# B&R Automation Studio project DuctLines
Automation Studio 4.2.14.119 SP

## Configuration DUCTO2_RIO

CPU X20CP1584, AutomationRuntime J4.25, Build 4.1.2, Vc V4.25.0, Safety 0.0

### Task classes (Cpu.sw)
```
Cyclic#1 (cycle 1000 us, tolerance 10000 us):
  IMotionCon <- IMotionControl.prg
  CleatRoll <- CleatRoll.prg
Cyclic#2 (cycle 10000 us, tolerance 20000 us):
  PDButtons <- PDButtons.prg
  Uncoiler_2 <- Uncoiler_2.prg
  CoilSelect <- CoilSelect.prg
  MarkTable <- MarkTable.prg
  MarkRF <- MarkRF.prg
  Feeder <- Feeder.prg
  SBrake <- SBrake.prg
  TDCTable <- TDCTable.prg
  TDCRFPshrs <- TDCRFPshrs.prg
  GlueApp <- GlueApp.prg
  Insulmatic <- Insulmatic.prg
  Pinspotter <- Pinspotter.prg
  BrakeCommo <- BrakeCommon.prg
  HydraulicB <- HydraulicBrakeCarriage.prg
  HWBwoPLC <- HWBwoPLC.prg
  MarkHead <- MarkHead.prg
Cyclic#4 (cycle 100000 us, tolerance 100000 us):
  HMIButtons <- HMIButtons.prg
  Server <- LibAsTCP1_ST.Server.prg
Binaries: TCData, arconfig, asfw, ashwd, iomap, User, Role, sysconf
Libraries: standard, MestekLib, AsTCP, runtime, asstring, asieccon, astime
```

### Hardware
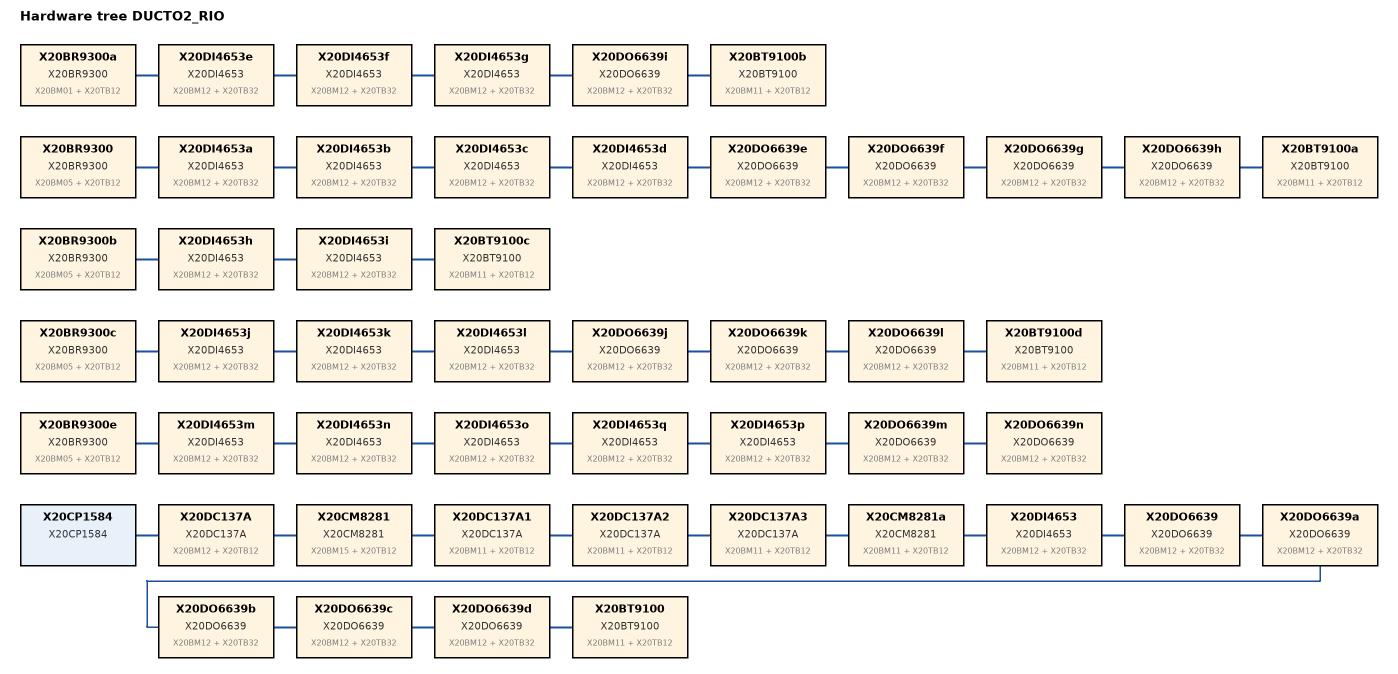
```
X20BM01 : X20BM01 v1.0.1.1
X20BM05 : X20BM05 v1.0.0.3
X20BM05b : X20BM05 v1.0.0.3
X20BM05c : X20BM05 v1.0.0.3
X20BM05d : X20BM05 v1.0.0.3
X20BM11 : X20BM11 v1.0.0.1  [X2X1 -> X20BM12f.X2X2]
X20BM11a : X20BM11 v1.0.0.1  [X2X1 -> X20BM11b.X2X2]
X20BM11b : X20BM11 v1.0.0.1  [X2X1 -> X20BM15.X2X2]
X20BM11c : X20BM11 v1.0.0.1  [X2X1 -> X20BM11a.X2X2]
X20BM11d : X20BM11 v1.0.0.1  [X2X1 -> X20BM11c.X2X2]
X20BM11e : X20BM11 v1.0.0.1  [X2X1 -> X20BM12n.X2X2]
X20BM11f : X20BM11 v1.0.0.1  [X2X1 -> X20BM12r.X2X2]
X20BM11g : X20BM11 v1.0.0.1  [X2X1 -> X20BM12t.X2X2]
X20BM11h : X20BM11 v1.0.0.1  [X2X1 -> X20BM12z.X2X2]
X20BM12 : X20BM12 v1.0.0.1  [X2X1 -> X20BM11d.X2X2]
X20BM12a : X20BM12 v1.0.0.1  [X2X1 -> X20CP1584.IF6]
X20BM12aa : X20BM12 v1.0.0.1  [X2X1 -> X20BM05d.X2X2]
X20BM12ab : X20BM12 v1.0.0.1  [X2X1 -> X20BM12aa.X2X2]
X20BM12ac : X20BM12 v1.0.0.1  [X2X1 -> X20BM12ab.X2X2]
X20BM12ad : X20BM12 v1.0.0.1  [X2X1 -> X20BM12ag.X2X2]
X20BM12ae : X20BM12 v1.0.0.1  [X2X1 -> X20BM12ad.X2X2]
X20BM12af : X20BM12 v1.0.0.1  [X2X1 -> X20BM12ae.X2X2]
X20BM12ag : X20BM12 v1.0.0.1  [X2X1 -> X20BM12ac.X2X2]
X20BM12b : X20BM12 v1.0.0.1  [X2X1 -> X20BM12.X2X2]
X20BM12c : X20BM12 v1.0.0.1  [X2X1 -> X20BM12b.X2X2]
X20BM12d : X20BM12 v1.0.0.1  [X2X1 -> X20BM12c.X2X2]
X20BM12e : X20BM12 v1.0.0.1  [X2X1 -> X20BM12d.X2X2]
X20BM12f : X20BM12 v1.0.0.1  [X2X1 -> X20BM12e.X2X2]
X20BM12g : X20BM12 v1.0.0.1  [X2X1 -> X20BM05.X2X2]
X20BM12h : X20BM12 v1.0.0.1  [X2X1 -> X20BM12g.X2X2]
X20BM12i : X20BM12 v1.0.0.1  [X2X1 -> X20BM12h.X2X2]
X20BM12j : X20BM12 v1.0.0.1  [X2X1 -> X20BM12i.X2X2]
X20BM12k : X20BM12 v1.0.0.1  [X2X1 -> X20BM12j.X2X2]
X20BM12l : X20BM12 v1.0.0.1  [X2X1 -> X20BM12k.X2X2]
X20BM12m : X20BM12 v1.0.0.1  [X2X1 -> X20BM12l.X2X2]
X20BM12n : X20BM12 v1.0.0.1  [X2X1 -> X20BM12m.X2X2]
X20BM12o : X20BM12 v1.0.0.1  [X2X1 -> X20BM01.X2X2]
X20BM12p : X20BM12 v1.0.0.1  [X2X1 -> X20BM12o.X2X2]
X20BM12q : X20BM12 v1.0.0.1  [X2X1 -> X20BM12p.X2X2]
X20BM12r : X20BM12 v1.0.0.1  [X2X1 -> X20BM12q.X2X2]
X20BM12s : X20BM12 v1.0.0.1  [X2X1 -> X20BM05b.X2X2]
X20BM12t : X20BM12 v1.0.0.1  [X2X1 -> X20BM12s.X2X2]
X20BM12u : X20BM12 v1.0.0.1  [X2X1 -> X20BM05c.X2X2]
X20BM12v : X20BM12 v1.0.0.1  [X2X1 -> X20BM12u.X2X2]
X20BM12w : X20BM12 v1.0.0.1  [X2X1 -> X20BM12v.X2X2]
X20BM12x : X20BM12 v1.0.0.1  [X2X1 -> X20BM12w.X2X2]
X20BM12y : X20BM12 v1.0.0.1  [X2X1 -> X20BM12x.X2X2]
X20BM12z : X20BM12 v1.0.0.1  [X2X1 -> X20BM12y.X2X2]
X20BM15 : X20BM15 v1.0.1.0  [X2X1 -> X20BM12a.X2X2 (NodeNumber=2)]
X20BR9300 : X20BR9300 v1.0.3.0  [SS1 -> X20TB12g.SS; SL -> X20BM05.SL1; X2X1 -> X20BT9100.X2X1 (NodeNumber=20)]
  Supervision = off
X20BR9300a : X20BR9300 v1.0.3.0  [SS1 -> X20TB12i.SS; SL -> X20BM01.SL1; X2X1 -> X20BT9100a.X2X1]
  Supervision = off
X20BR9300b : X20BR9300 v1.0.3.0  [SS1 -> X20TB12k.SS; SL -> X20BM05b.SL1; X2X1 -> X20BT9100b.X2X1 (NodeNumber=40)]
  Supervision = off
X20BR9300c : X20BR9300 v1.0.3.0  [SS1 -> X20TB12m.SS; SL -> X20BM05c.SL1; X2X1 -> X20BT9100c.X2X1 (NodeNumber=50)]
  Supervision = off
X20BR9300e : X20BR9300 v1.0.3.0  [SS1 -> X20TB12p.SS; SL -> X20BM05d.SL1; X2X1 -> X20BT9100d.X2X1 (NodeNumber=60)]
  Supervision = off
X20BT9100 : X20BT9100 v1.0.2.4  [SS1 -> X20TB12f.SS; SL -> X20BM11.SL1]
  Supervision = off
X20BT9100a : X20BT9100 v1.0.2.4  [SS1 -> X20TB12h.SS; SL -> X20BM11e.SL1]
  Supervision = off
X20BT9100b : X20BT9100 v1.0.2.4  [SS1 -> X20TB12j.SS; SL -> X20BM11f.SL1]
  Supervision = off
X20BT9100c : X20BT9100 v1.0.2.4  [SS1 -> X20TB12l.SS; SL -> X20BM11g.SL1]
  Supervision = off
X20BT9100d : X20BT9100 v1.0.2.4  [SS1 -> X20TB12n.SS; SL -> X20BM11h.SL1]
  Supervision = off
X20CM8281 : X20CM8281 v1.0.4.0  [SS1 -> X20TB12.SS; SL -> X20BM15.SL1]
  Supervision = off
X20CM8281a : X20CM8281 v1.0.4.0  [SS1 -> X20TB12e.SS; SL -> X20BM11d.SL1]
  Supervision = off
X20CP1584 : X20CP1584 v1.3.0.0
  Connector IF2:
    ActivateDevice = 1
    EthInterfaceRedundant = 0
    Mode = Manual
    InternetAddress = 10.1.254.101
  Connector IF3:
    EplInterfaceRedundant = 0
    EplEthInterfaceRedundant = 0
  ConfigurationID = X20_CPU_test
  EnableUsbRemoteInstall = 1
  TimerDeviceType = SWIOTIMER
  Cyclic1Duration = 1000
  Cyclic1Tolerance = 10000
  Cyclic2Duration = 10000
  Cyclic2Tolerance = 20000
  Cyclic3Duration = 50000
  Cyclic3Tolerance = 50000
  Cyclic4Duration = 100000
  Cyclic4Tolerance = 100000
  Cyclic5Duration = 200000
  Cyclic5Tolerance = 200000
  Cyclic6Duration = 500000
  Cyclic6Tolerance = 500000
  Cyclic7Duration = 1000000
  Cyclic7Tolerance = 1000000
  Cyclic8Duration = 10000
  Cyclic8Tolerance = 30000000
X20DC137A : X20DC137A v1.0.0.3 (LastFrozenVersion=1.0.0.3)  [SS1 -> X20TB12b.SS; SL -> X20BM12a.SL1]
  Supervision = off
  CounterStd01 = 32Bit
  BWConfigChannel03 = off
X20DC137A1 : X20DC137A v1.0.0.3 (LastFrozenVersion=1.0.0.3)  [SS1 -> X20TB12c.SS; SL -> X20BM11b.SL1]
  Supervision = off
  CounterStd01 = 32Bit
  BWConfigChannel03 = off
X20DC137A2 : X20DC137A v1.0.0.3 (LastFrozenVersion=1.0.0.3)  [SS1 -> X20TB12a.SS; SL -> X20BM11a.SL1]
  Supervision = off
  CounterStd01 = 32Bit
  BWConfigChannel03 = off
X20DC137A3 : X20DC137A v1.0.0.3 (LastFrozenVersion=1.0.0.3)  [SS1 -> X20TB12d.SS; SL -> X20BM11c.SL1]
  Supervision = off
  CounterStd01 = 32Bit
  BWConfigChannel03 = off
X20DI4653 : X20DI4653 v1.0.2.0  [SS1 -> X20TB32.SS; SL -> X20BM12.SL1]
  Supervision = off
X20DI4653a : X20DI4653 v1.0.2.0  [SS1 -> X20TB32f.SS; SL -> X20BM12g.SL1]
  Supervision = off
X20DI4653b : X20DI4653 v1.0.2.0  [SS1 -> X20TB32g.SS; SL -> X20BM12h.SL1]
  Supervision = off
X20DI4653c : X20DI4653 v1.0.2.0  [SS1 -> X20TB32h.SS; SL -> X20BM12i.SL1]
  Supervision = off
X20DI4653d : X20DI4653 v1.0.2.0  [SS1 -> X20TB32i.SS; SL -> X20BM12j.SL1]
  Supervision = off
X20DI4653e : X20DI4653 v1.0.2.0  [SS1 -> X20TB32n.SS; SL -> X20BM12o.SL1]
  Supervision = off
X20DI4653f : X20DI4653 v1.0.2.0  [SS1 -> X20TB32o.SS; SL -> X20BM12p.SL1]
  Supervision = off
X20DI4653g : X20DI4653 v1.0.2.0  [SS1 -> X20TB32p.SS; SL -> X20BM12q.SL1]
  Supervision = off
X20DI4653h : X20DI4653 v1.0.2.0  [SS1 -> X20TB32r.SS; SL -> X20BM12s.SL1]
  Supervision = off
X20DI4653i : X20DI4653 v1.0.2.0  [SS1 -> X20TB32s.SS; SL -> X20BM12t.SL1]
  Supervision = off
X20DI4653j : X20DI4653 v1.0.2.0  [SS1 -> X20TB32t.SS; SL -> X20BM12u.SL1]
  Supervision = off
X20DI4653k : X20DI4653 v1.0.2.0  [SS1 -> X20TB32u.SS; SL -> X20BM12v.SL1]
  Supervision = off
X20DI4653l : X20DI4653 v1.0.2.0  [SS1 -> X20TB32v.SS; SL -> X20BM12w.SL1]
  Supervision = off
X20DI4653m : X20DI4653 v1.0.2.0  [SS1 -> X20TB32z.SS; SL -> X20BM12aa.SL1]
  Supervision = off
X20DI4653n : X20DI4653 v1.0.2.0  [SS1 -> X20TB32aa.SS; SL -> X20BM12ab.SL1]
  Supervision = off
X20DI4653o : X20DI4653 v1.0.2.0  [SS1 -> X20TB32ab.SS; SL -> X20BM12ac.SL1]
  Supervision = off
X20DI4653p : X20DI4653 v1.0.2.0  [SS1 -> X20TB32ac.SS; SL -> X20BM12ad.SL1]
  Supervision = off
X20DI4653q : X20DI4653 v1.0.2.0  [SS1 -> X20TB32af.SS; SL -> X20BM12ag.SL1]
  Supervision = off
X20DO6639 : X20DO6639 v1.0.1.0  [SS1 -> X20TB32a.SS; SL -> X20BM12b.SL1]
  Supervision = off
X20DO6639a : X20DO6639 v1.0.1.0  [SS1 -> X20TB32b.SS; SL -> X20BM12c.SL1]
  Supervision = off
X20DO6639b : X20DO6639 v1.0.1.0  [SS1 -> X20TB32c.SS; SL -> X20BM12d.SL1]
  Supervision = off
X20DO6639c : X20DO6639 v1.0.1.0  [SS1 -> X20TB32d.SS; SL -> X20BM12e.SL1]
  Supervision = off
X20DO6639d : X20DO6639 v1.0.1.0  [SS1 -> X20TB32e.SS; SL -> X20BM12f.SL1]
  Supervision = off
X20DO6639e : X20DO6639 v1.0.1.0  [SS1 -> X20TB32j.SS; SL -> X20BM12k.SL1]
  Supervision = off
X20DO6639f : X20DO6639 v1.0.1.0  [SS1 -> X20TB32k.SS; SL -> X20BM12l.SL1]
  Supervision = off
X20DO6639g : X20DO6639 v1.0.1.0  [SS1 -> X20TB32l.SS; SL -> X20BM12m.SL1]
  Supervision = off
X20DO6639h : X20DO6639 v1.0.1.0  [SS1 -> X20TB32m.SS; SL -> X20BM12n.SL1]
  Supervision = off
X20DO6639i : X20DO6639 v1.0.1.0  [SS1 -> X20TB32q.SS; SL -> X20BM12r.SL1]
  Supervision = off
X20DO6639j : X20DO6639 v1.0.1.0  [SS1 -> X20TB32w.SS; SL -> X20BM12x.SL1]
  Supervision = off
X20DO6639k : X20DO6639 v1.0.1.0  [SS1 -> X20TB32x.SS; SL -> X20BM12y.SL1]
  Supervision = off
X20DO6639l : X20DO6639 v1.0.1.0  [SS1 -> X20TB32y.SS; SL -> X20BM12z.SL1]
  Supervision = off
X20DO6639m : X20DO6639 v1.0.1.0  [SS1 -> X20TB32ad.SS; SL -> X20BM12ae.SL1]
  Supervision = off
X20DO6639n : X20DO6639 v1.0.1.0  [SS1 -> X20TB32ae.SS; SL -> X20BM12af.SL1]
  Supervision = off
X20TB12 : X20TB12 v1.0.0.0
X20TB12a : X20TB12 v1.0.0.0
X20TB12b : X20TB12 v1.0.0.0
X20TB12c : X20TB12 v1.0.0.0
X20TB12d : X20TB12 v1.0.0.0
X20TB12e : X20TB12 v1.0.0.0
X20TB12f : X20TB12 v1.0.0.0
X20TB12g : X20TB12 v1.0.0.0
X20TB12h : X20TB12 v1.0.0.0
X20TB12i : X20TB12 v1.0.0.0
X20TB12j : X20TB12 v1.0.0.0
X20TB12k : X20TB12 v1.0.0.0
X20TB12l : X20TB12 v1.0.0.0
X20TB12m : X20TB12 v1.0.0.0
X20TB12n : X20TB12 v1.0.0.0
X20TB12p : X20TB12 v1.0.0.0
X20TB32 : X20TB32 v1.0.0.1
X20TB32a : X20TB32 v1.0.0.1
X20TB32aa : X20TB32 v1.0.0.1
X20TB32ab : X20TB32 v1.0.0.1
X20TB32ac : X20TB32 v1.0.0.1
X20TB32ad : X20TB32 v1.0.0.1
X20TB32ae : X20TB32 v1.0.0.1
X20TB32af : X20TB32 v1.0.0.1
X20TB32b : X20TB32 v1.0.0.1
X20TB32c : X20TB32 v1.0.0.1
X20TB32d : X20TB32 v1.0.0.1
X20TB32e : X20TB32 v1.0.0.1
X20TB32f : X20TB32 v1.0.0.1
X20TB32g : X20TB32 v1.0.0.1
X20TB32h : X20TB32 v1.0.0.1
X20TB32i : X20TB32 v1.0.0.1
X20TB32j : X20TB32 v1.0.0.1
X20TB32k : X20TB32 v1.0.0.1
X20TB32l : X20TB32 v1.0.0.1
X20TB32m : X20TB32 v1.0.0.1
X20TB32n : X20TB32 v1.0.0.1
X20TB32o : X20TB32 v1.0.0.1
X20TB32p : X20TB32 v1.0.0.1
X20TB32q : X20TB32 v1.0.0.1
X20TB32r : X20TB32 v1.0.0.1
X20TB32s : X20TB32 v1.0.0.1
X20TB32t : X20TB32 v1.0.0.1
X20TB32u : X20TB32 v1.0.0.1
X20TB32v : X20TB32 v1.0.0.1
X20TB32w : X20TB32 v1.0.0.1
X20TB32x : X20TB32 v1.0.0.1
X20TB32y : X20TB32 v1.0.0.1
X20TB32z : X20TB32 v1.0.0.1
```

### IoMap.iom - X20CP1584/IoMap.iom
```iecst
VAR_CONFIG
	Cyclic#1.ActlMetalEncoder AT %ID."X20DC137A".Encoder01;
	Cyclic#1.::ProcessorEncoderReset AT %QX."X20DC137A".Encoder01Reset;
	Cyclic#1.ActualDAC1 AT %QW."X20CM8281".AnalogOutput01;
	Cyclic#1.ElectricDriveEnable AT %QX."X20CM8281".DigitalOutput01;
	Cyclic#2.MarkEncoderResetSignal AT %QX."X20DC137A1".Encoder01Reset;
	Cyclic#2.RawMarkEncoder AT %ID."X20DC137A1".Encoder01;
	Cyclic#2.PinspotEncoder AT %ID."X20DC137A2".Encoder01;
	Cyclic#2.PinspotEncoderResetSignal AT %QX."X20DC137A2".Encoder01Reset;
	Cyclic#2.::BrakeEncoderReset AT %QX."X20DC137A3".Encoder01Reset;
	Cyclic#2.BrakeEncoder AT %ID."X20DC137A3".Encoder01;
	Cyclic#2.EStopClear AT %IX."X20DI4653".DigitalInput01;
	Cyclic#2.::PowerOn AT %IX."X20DI4653".DigitalInput02;
	Cyclic#2.doCoilSelect AT %QX."X20DO6639".DigitalOutput01;
	Cyclic#2.doProDuctHydraulics AT %QX."X20DO6639".DigitalOutput02;
	Cyclic#2.BrakeHydraulics AT %QX."X20DO6639".DigitalOutput03;
	Cyclic#2.::MarkTableFwd AT %QX."X20DO6639".DigitalOutput04;
	Cyclic#2.::MarkPshrFwd AT %QX."X20DO6639".DigitalOutput05;
	Cyclic#2.::MarkPusherReverse AT %QX."X20DO6639".DigitalOutput06;
	Cyclic#2.::MarkRollformerOn AT %QX."X20DO6639a".DigitalOutput01;
	Cyclic#2.::TDCConveyorRun AT %QX."X20DO6639a".DigitalOutput02;
	Cyclic#2.::TDCTablePusherFwd AT %QX."X20DO6639a".DigitalOutput03;
	Cyclic#2.::TDCTablePusherReverse AT %QX."X20DO6639a".DigitalOutput04;
	Cyclic#2.doTDCAdjustableHeadIn AT %QX."X20DO6639a".DigitalOutput05;
	Cyclic#2.doTDCAdjustableHeadOut AT %QX."X20DO6639a".DigitalOutput06;
	Cyclic#2.doTDCFixedHeadIn AT %QX."X20DO6639b".DigitalOutput01;
	Cyclic#2.doTDCFixedHeadOut AT %QX."X20DO6639b".DigitalOutput02;
	Cyclic#2.::TDCRFMotor AT %QX."X20DO6639b".DigitalOutput03;
	Cyclic#2.::TDCRFPusherFwd AT %QX."X20DO6639b".DigitalOutput04;
	Cyclic#2.::TDCRFPusherRev AT %QX."X20DO6639b".DigitalOutput05;
	Cyclic#2.::InsulmaticEntranceLowSpeed AT %QX."X20DO6639c".DigitalOutput01;
	Cyclic#2.::InsulmaticExitLowSpeed AT %QX."X20DO6639c".DigitalOutput02;
	Cyclic#2.::InsulmaticExitHiSpeed AT %QX."X20DO6639c".DigitalOutput03;
	Cyclic#2.::InsulmaticEntranceHiSpeed AT %QX."X20DO6639c".DigitalOutput04;
	Cyclic#2.::BrakeConveyorLow AT %QX."X20DO6639c".DigitalOutput05;
	Cyclic#2.::BrakeConveyorHigh AT %QX."X20DO6639c".DigitalOutput06;
	Cyclic#2.::AmberLight AT %QX."X20DO6639d".DigitalOutput01;
	Cyclic#2.::BlueLight AT %QX."X20DO6639d".DigitalOutput02;
	Cyclic#2.::WarningHorn AT %QX."X20DO6639d".DigitalOutput03;
	Cyclic#2.::MarkTableRev AT %QX."X20DO6639d".DigitalOutput04;
	Cyclic#2.::UncoilerJogForwardPB AT %IX."X20DI4653a".DigitalInput01;
	Cyclic#2.::UncoilerJogReversePB AT %IX."X20DI4653a".DigitalInput02;
	Cyclic#2.::SlackBar AT %IX."X20DI4653a".DigitalInput03;
	Cyclic#2.diCoilSelectJog AT %IX."X20DI4653a".DigitalInput04;
	Cyclic#2.::ProcessorJogFwd AT %IX."X20DI4653b".DigitalInput01;
	Cyclic#2.::ProcessorJogRev AT %IX."X20DI4653b".DigitalInput02;
	Cyclic#2.::MatlAtMeasureRoll AT %IX."X20DI4653b".DigitalInput03;
	Cyclic#2.::ShearClampDownProx AT %IX."X20DI4653c".DigitalInput01;
	Cyclic#2.::ShearClampUpProx AT %IX."X20DI4653c".DigitalInput02;
	Cyclic#2.::ShearLeafDownProx AT %IX."X20DI4653c".DigitalInput03;
	Cyclic#2.::ShearLeafUpProx AT %IX."X20DI4653c".DigitalInput04;
	Cyclic#2.::HumpLimitSwitch AT %IX."X20DI4653d".DigitalInput01;
	Cyclic#2.::ShearValve AT %QX."X20DO6639e".DigitalOutput01;
	Cyclic#2.::VValve AT %QX."X20DO6639e".DigitalOutput02;
	Cyclic#2.::LTValve AT %QX."X20DO6639e".DigitalOutput04;
	Cyclic#2.::CenterShuttleOutput AT %QX."X20DO6639e".DigitalOutput05;
	Cyclic#2.::CHoleValve AT %QX."X20DO6639e".DigitalOutput06;
	Cyclic#2.::LeftShuttleOutput AT %QX."X20DO6639f".DigitalOutput01;
	Cyclic#2.::LHoleValve AT %QX."X20DO6639f".DigitalOutput02;
	Cyclic#2.::RightShuttleOutput AT %QX."X20DO6639f".DigitalOutput03;
	Cyclic#2.::RHoleValve AT %QX."X20DO6639f".DigitalOutput04;
	Cyclic#2.::LeftKnockDownRoll AT %QX."X20DO6639f".DigitalOutput05;
	Cyclic#2.::RightKnockDownRoll AT %QX."X20DO6639f".DigitalOutput06;
	Cyclic#2.::ShearClampLowerSolenoid AT %QX."X20DO6639g".DigitalOutput01;
	Cyclic#2.::ShearClampRaiseSolenoid AT %QX."X20DO6639g".DigitalOutput02;
	Cyclic#2.::ShearLeafLowerSolenoid AT %QX."X20DO6639g".DigitalOutput03;
	Cyclic#2.::ShearLeafRaiseSolenoid AT %QX."X20DO6639g".DigitalOutput04;
	Cyclic#2.::SnapLockButtonGag AT %QX."X20DO6639h".DigitalOutput01;
	Cyclic#2.doCoilSelectRollClose AT %QX."X20DO6639h".DigitalOutput02;
	Cyclic#2.::UncoilerRun AT %QX."X20DO6639h".DigitalOutput03;
	Cyclic#2.::UncoilerForwardSolenoid AT %QX."X20DO6639h".DigitalOutput04;
	Cyclic#2.::UncoilerReverseSolenoid AT %QX."X20DO6639h".DigitalOutput05;
	Cyclic#2.diFeedInitButton AT %IX."X20DI4653f".DigitalInput01;
	Cyclic#2.::TDCTablePartProx AT %IX."X20DI4653f".DigitalInput02;
	Cyclic#2.::TDCTablePause AT %IX."X20DI4653f".DigitalInput03;
	Cyclic#2.::TDCTablePushStop AT %IX."X20DI4653f".DigitalInput04;
	Cyclic#2.::TDCTablePusherRevPB AT %IX."X20DI4653g".DigitalInput01;
	Cyclic#2.::diMarkHeadUpProx AT %IX."X20DI4653g".DigitalInput02;
	Cyclic#2.::diMarkHeadDownProx AT %IX."X20DI4653g".DigitalInput03;
	Cyclic#2.::MarkGateRaise AT %QX."X20DO6639i".DigitalOutput01;
	Cyclic#2.doMarkRollformerHeadLower AT %QX."X20DO6639i".DigitalOutput02;
	Cyclic#2.doMarkRollformerHeadRaise AT %QX."X20DO6639i".DigitalOutput03;
	Cyclic#2.diTDCFixedHeadJogIn AT %IX."X20DI4653h".DigitalInput01;
	Cyclic#2.diTDCFixedHeadJogOut AT %IX."X20DI4653h".DigitalInput02;
	Cyclic#2.diTDCAdjustableHeadJogIn AT %IX."X20DI4653h".DigitalInput03;
	Cyclic#2.diTDCAdjustableHeadJogOut AT %IX."X20DI4653h".DigitalInput04;
	Cyclic#2.::diTDCRollformerJog AT %IX."X20DI4653i".DigitalInput01;
	Cyclic#2.::TDCPushStrokeComplete AT %IX."X20DI4653i".DigitalInput03;
	Cyclic#2.::TDCPusherRevPB AT %IX."X20DI4653i".DigitalInput04;
	Cyclic#2.::GluePartSense AT %IX."X20DI4653j".DigitalInput01;
	Cyclic#2.::RaiseImaticBlade AT %IX."X20DI4653k".DigitalInput01;
	Cyclic#2.::InsulationFeed AT %IX."X20DI4653k".DigitalInput02;
	Cyclic#2.::ISquarePinOn AT %IX."X20DI4653k".DigitalInput03;
	Cyclic#2.::PartAtISquarePin AT %IX."X20DI4653k".DigitalInput04;
	Cyclic#2.::PartAtInsulationFeed AT %IX."X20DI4653l".DigitalInput01;
	Cyclic#2.::PartPresentPSpotter AT %IX."X20DI4653l".DigitalInput02;
	Cyclic#2.::GlueSprayEnable AT %QX."X20DO6639j".DigitalOutput03;
	Cyclic#2.::ImaticFeedRoll AT %QX."X20DO6639k".DigitalOutput03;
	Cyclic#2.::ImaticPressRoll AT %QX."X20DO6639k".DigitalOutput04;
	Cyclic#2.::ImaticSquarePin AT %QX."X20DO6639k".DigitalOutput05;
	Cyclic#2.::ImaticBladeUp AT %QX."X20DO6639l".DigitalOutput01;
	Cyclic#2.::ImaticBladeDown AT %QX."X20DO6639l".DigitalOutput02;
	Cyclic#2.::PinspotterDrive AT %QX."X20DO6639l".DigitalOutput03;
	Cyclic#2.::CarriageReference AT %IX."X20DI4653m".DigitalInput01;
	Cyclic#2.::BrakeArmLwrInhibit AT %IX."X20DI4653m".DigitalInput02;
	Cyclic#2.::BrakeBeamLwrInhibit AT %IX."X20DI4653m".DigitalInput03;
	Cyclic#2.::EjectComplete AT %IX."X20DI4653m".DigitalInput04;
	Cyclic#2.::BrakeLeafHomeProx AT %IX."X20DI4653n".DigitalInput01;
	Cyclic#2.::BrakeBeamDownProx AT %IX."X20DI4653n".DigitalInput02;
	Cyclic#2.::BrakeBeamUpProx AT %IX."X20DI4653n".DigitalInput03;
	Cyclic#2.diWBrakeArmsUp AT %IX."X20DI4653n".DigitalInput04;
	Cyclic#2.::BrakePartPresent AT %IX."X20DI4653o".DigitalInput01;
	Cyclic#2.::MaterialClamped AT %IX."X20DI4653o".DigitalInput02;
	Cyclic#2.BrakeManualButton AT %IX."X20DI4653o".DigitalInput04;
	Cyclic#2.::BrakeSingleCycle AT %IX."X20DI4653p".DigitalInput01;
	Cyclic#2.::MoveToBeam AT %QX."X20DO6639m".DigitalOutput01;
	Cyclic#2.::MoveAwayBeam AT %QX."X20DO6639m".DigitalOutput02;
	Cyclic#2.::BrakeHighSpeedRelay AT %QX."X20DO6639m".DigitalOutput03;
	Cyclic#2.::CarriageArmRaise AT %QX."X20DO6639m".DigitalOutput04;
	Cyclic#2.::CarriageArmLower AT %QX."X20DO6639m".DigitalOutput05;
	Cyclic#2.::CarriageClampClose AT %QX."X20DO6639m".DigitalOutput06;
	Cyclic#2.::BrakeBeamRaise AT %QX."X20DO6639n".DigitalOutput01;
	Cyclic#2.::BrakeBeamLower AT %QX."X20DO6639n".DigitalOutput02;
	Cyclic#2.::BrakeLeafRaise AT %QX."X20DO6639n".DigitalOutput03;
	Cyclic#2.::BrakeLeafLower AT %QX."X20DO6639n".DigitalOutput04;
	Cyclic#2.::BrakeManualIndicator AT %QX."X20DO6639n".DigitalOutput05;
	Cyclic#2.::BrakeAutoIndicator AT %QX."X20DO6639n".DigitalOutput06;
	Cyclic#2.::BrakeAutoButton AT %IX."X20DI4653q".DigitalInput01;
	Cyclic#2.diBrakeCarriageJogIn AT %IX."X20DI4653q".DigitalInput02;
	Cyclic#2.diBrakeCarriageJogOut AT %IX."X20DI4653q".DigitalInput03;
	Cyclic#2.::BrakeSequenceReset AT %IX."X20DI4653q".DigitalInput04;
	Cyclic#2.::MatlAtMarkTable AT %IX."X20DI4653e".DigitalInput01;
	Cyclic#2.::MarkPushComplete AT %IX."X20DI4653e".DigitalInput02;
	Cyclic#2.::MarkPusherStop AT %IX."X20DI4653e".DigitalInput03;
	Cyclic#2.::MarkTTPusherJogRevPB AT %IX."X20DI4653e".DigitalInput04;
END_VAR
```

## Configuration DUCTO2_V02

CPU X20CP1584, AutomationRuntime J4.25, Build 4.1.2, Vc V4.25.0, Safety 0.0

### Hardware
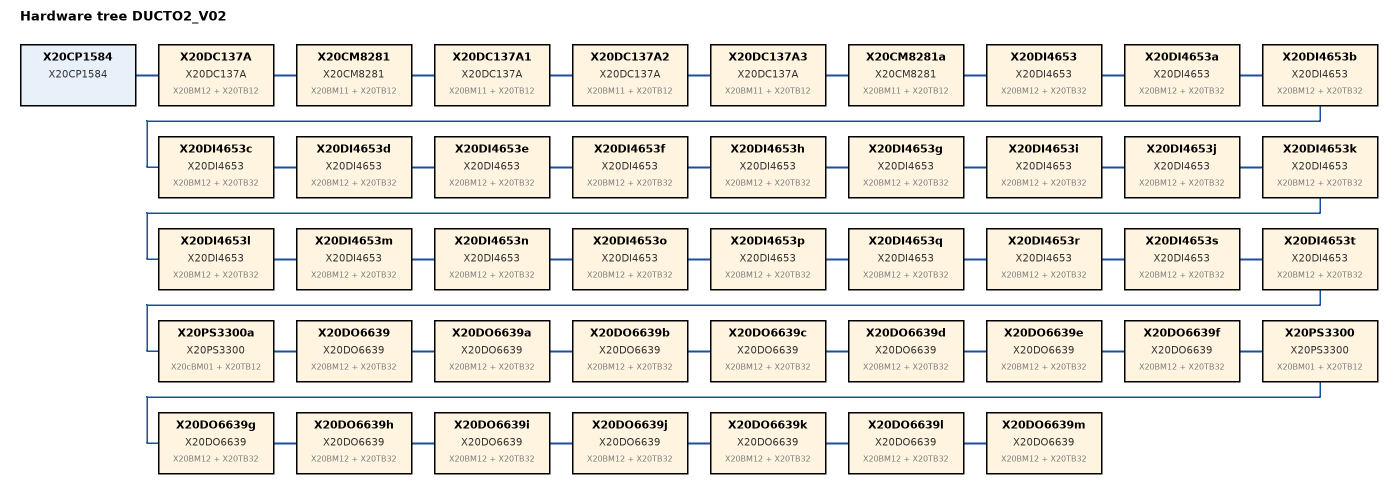
```
X20BM01 : X20BM01 v1.0.1.1  [X2X1 -> X20BM12ab.X2X2]
X20BM11 : X20BM11 v1.0.0.1  [X2X1 -> X20BM12a.X2X2]
X20BM11a : X20BM11 v1.0.0.1  [X2X1 -> X20BM11b.X2X2]
X20BM11b : X20BM11 v1.0.0.1  [X2X1 -> X20BM11.X2X2]
X20BM11c : X20BM11 v1.0.0.1  [X2X1 -> X20BM11a.X2X2]
X20BM11d : X20BM11 v1.0.0.1  [X2X1 -> X20BM11c.X2X2]
X20BM12 : X20BM12 v1.0.0.1  [X2X1 -> X20BM11d.X2X2]
X20BM12a : X20BM12 v1.0.0.1  [X2X1 -> X20CP1584.IF6]
X20BM12aa : X20BM12 v1.0.0.1  [X2X1 -> X20BM12z.X2X2]
X20BM12ab : X20BM12 v1.0.0.1  [X2X1 -> X20BM12aa.X2X2]
X20BM12ac : X20BM12 v1.0.0.1  [X2X1 -> X20BM01.X2X2]
X20BM12ad : X20BM12 v1.0.0.1  [X2X1 -> X20BM12ac.X2X2]
X20BM12ae : X20BM12 v1.0.0.1  [X2X1 -> X20BM12ad.X2X2]
X20BM12af : X20BM12 v1.0.0.1  [X2X1 -> X20BM12ae.X2X2]
X20BM12ag : X20BM12 v1.0.0.1  [X2X1 -> X20BM12af.X2X2]
X20BM12ah : X20BM12 v1.0.0.1  [X2X1 -> X20BM12ag.X2X2]
X20BM12ai : X20BM12 v1.0.0.1  [X2X1 -> X20BM12ah.X2X2]
X20BM12b : X20BM12 v1.0.0.1  [X2X1 -> X20BM12.X2X2]
X20BM12c : X20BM12 v1.0.0.1  [X2X1 -> X20BM12b.X2X2]
X20BM12d : X20BM12 v1.0.0.1  [X2X1 -> X20BM12c.X2X2]
X20BM12e : X20BM12 v1.0.0.1  [X2X1 -> X20BM12d.X2X2]
X20BM12f : X20BM12 v1.0.0.1  [X2X1 -> X20BM12e.X2X2]
X20BM12g : X20BM12 v1.0.0.1  [X2X1 -> X20BM12f.X2X2]
X20BM12h : X20BM12 v1.0.0.1  [X2X1 -> X20BM12i.X2X2]
X20BM12i : X20BM12 v1.0.0.1  [X2X1 -> X20BM12g.X2X2]
X20BM12j : X20BM12 v1.0.0.1  [X2X1 -> X20BM12h.X2X2]
X20BM12k : X20BM12 v1.0.0.1  [X2X1 -> X20BM12j.X2X2]
X20BM12l : X20BM12 v1.0.0.1  [X2X1 -> X20BM12k.X2X2]
X20BM12m : X20BM12 v1.0.0.1  [X2X1 -> X20BM12l.X2X2]
X20BM12n : X20BM12 v1.0.0.1  [X2X1 -> X20BM12m.X2X2]
X20BM12o : X20BM12 v1.0.0.1  [X2X1 -> X20BM12n.X2X2]
X20BM12p : X20BM12 v1.0.0.1  [X2X1 -> X20BM12o.X2X2]
X20BM12q : X20BM12 v1.0.0.1  [X2X1 -> X20BM12p.X2X2]
X20BM12r : X20BM12 v1.0.0.1  [X2X1 -> X20BM12q.X2X2]
X20BM12s : X20BM12 v1.0.0.1  [X2X1 -> X20BM12r.X2X2]
X20BM12t : X20BM12 v1.0.0.1  [X2X1 -> X20BM12s.X2X2]
X20BM12u : X20BM12 v1.0.0.1  [X2X1 -> X20BM12t.X2X2]
X20BM12v : X20BM12 v1.0.0.1  [X2X1 -> X20cBM01.X2X2]
X20BM12w : X20BM12 v1.0.0.1  [X2X1 -> X20BM12v.X2X2]
X20BM12x : X20BM12 v1.0.0.1  [X2X1 -> X20BM12w.X2X2]
X20BM12y : X20BM12 v1.0.0.1  [X2X1 -> X20BM12x.X2X2]
X20BM12z : X20BM12 v1.0.0.1  [X2X1 -> X20BM12y.X2X2]
X20CM8281 : X20CM8281 v1.0.4.0  [SS1 -> X20TB12.SS; SL -> X20BM11.SL1]
  Supervision = off
X20CM8281a : X20CM8281 v1.0.4.0  [SS1 -> X20TB12e.SS; SL -> X20BM11d.SL1]
  Supervision = off
X20CP1584 : X20CP1584 v1.3.0.0
  Connector IF2:
    ActivateDevice = 1
    EthInterfaceRedundant = 0
    Mode = Manual
    InternetAddress = 10.1.254.101
  Connector IF3:
    EplInterfaceRedundant = 0
    CycleTime = 1000
    EplEthInterfaceRedundant = 0
  Connector IF6:
    CycleTime = 1000
  ConfigurationID = X20_CPU_test
  PermanentPvSize = 4096
  EnableUsbRemoteInstall = 1
  TimerDeviceType = EPLX2X
  Cyclic1Duration = 1000
  Cyclic1Tolerance = 0
  Cyclic1Output = 1
  Cyclic2Duration = 20000
  Cyclic2Tolerance = 20000
  Cyclic3Duration = 50000
  Cyclic3Tolerance = 50000
  Cyclic4Duration = 100000
  Cyclic4Tolerance = 100000
  Cyclic5Duration = 200000
  Cyclic5Tolerance = 200000
  Cyclic6Duration = 500000
  Cyclic6Tolerance = 500000
  Cyclic7Duration = 1000000
  Cyclic7Tolerance = 1000000
  Cyclic8Duration = 10000
  Cyclic8Tolerance = 30000000
  TimerDevice = X20CP1584.IF6
X20DC137A : X20DC137A v1.0.0.3  [SS1 -> X20TB12b.SS; SL -> X20BM12a.SL1]
  Supervision = off
  CounterStd01 = 32Bit
  BWConfigChannel03 = off
X20DC137A1 : X20DC137A v1.0.0.3  [SS1 -> X20TB12c.SS; SL -> X20BM11b.SL1]
  Supervision = off
  CounterStd01 = 32Bit
  BWConfigChannel03 = off
X20DC137A2 : X20DC137A v1.0.0.3  [SS1 -> X20TB12a.SS; SL -> X20BM11a.SL1]
  Supervision = off
  CounterStd01 = 32Bit
  BWConfigChannel03 = off
X20DC137A3 : X20DC137A v1.0.0.3  [SS1 -> X20TB12d.SS; SL -> X20BM11c.SL1]
  Supervision = off
  CounterStd01 = 32Bit
  BWConfigChannel03 = off
X20DI4653 : X20DI4653 v1.0.2.0  [SS1 -> X20TB32.SS; SL -> X20BM12.SL1]
  Supervision = off
X20DI4653a : X20DI4653 v1.0.2.0  [SS1 -> X20TB32a.SS; SL -> X20BM12b.SL1]
  Supervision = off
X20DI4653b : X20DI4653 v1.0.2.0  [SS1 -> X20TB32b.SS; SL -> X20BM12c.SL1]
  Supervision = off
X20DI4653c : X20DI4653 v1.0.2.0  [SS1 -> X20TB32c.SS; SL -> X20BM12d.SL1]
  Supervision = off
X20DI4653d : X20DI4653 v1.0.2.0  [SS1 -> X20TB32d.SS; SL -> X20BM12e.SL1]
  Supervision = off
X20DI4653e : X20DI4653 v1.0.2.0  [SS1 -> X20TB32e.SS; SL -> X20BM12f.SL1]
  Supervision = off
X20DI4653f : X20DI4653 v1.0.2.0  [SS1 -> X20TB32f.SS; SL -> X20BM12g.SL1]
  Supervision = off
X20DI4653g : X20DI4653 v1.0.2.0  [SS1 -> X20TB32g.SS; SL -> X20BM12h.SL1]
  Supervision = off
X20DI4653h : X20DI4653 v1.0.2.0  [SS1 -> X20TB32h.SS; SL -> X20BM12i.SL1]
  Supervision = off
X20DI4653i : X20DI4653 v1.0.2.0  [SS1 -> X20TB32i.SS; SL -> X20BM12j.SL1]
  Supervision = off
X20DI4653j : X20DI4653 v1.0.2.0  [SS1 -> X20TB32j.SS; SL -> X20BM12k.SL1]
  Supervision = off
X20DI4653k : X20DI4653 v1.0.2.0  [SS1 -> X20TB32k.SS; SL -> X20BM12l.SL1]
  Supervision = off
X20DI4653l : X20DI4653 v1.0.2.0  [SS1 -> X20TB32l.SS; SL -> X20BM12m.SL1]
  Supervision = off
X20DI4653m : X20DI4653 v1.0.2.0  [SS1 -> X20TB32m.SS; SL -> X20BM12n.SL1]
  Supervision = off
X20DI4653n : X20DI4653 v1.0.2.0  [SS1 -> X20TB32n.SS; SL -> X20BM12o.SL1]
  Supervision = off
X20DI4653o : X20DI4653 v1.0.2.0  [SS1 -> X20TB32o.SS; SL -> X20BM12p.SL1]
  Supervision = off
X20DI4653p : X20DI4653 v1.0.2.0  [SS1 -> X20TB32p.SS; SL -> X20BM12q.SL1]
  Supervision = off
X20DI4653q : X20DI4653 v1.0.2.0  [SS1 -> X20TB32q.SS; SL -> X20BM12r.SL1]
  Supervision = off
X20DI4653r : X20DI4653 v1.0.2.0  [SS1 -> X20TB32r.SS; SL -> X20BM12s.SL1]
  Supervision = off
X20DI4653s : X20DI4653 v1.0.2.0  [SS1 -> X20TB32s.SS; SL -> X20BM12t.SL1]
  Supervision = off
X20DI4653t : X20DI4653 v1.0.2.0  [SS1 -> X20TB32t.SS; SL -> X20BM12u.SL1]
  Supervision = off
X20DO6639 : X20DO6639 v1.0.1.0  [SS1 -> X20TB32u.SS; SL -> X20BM12v.SL1]
  Supervision = off
X20DO6639a : X20DO6639 v1.0.1.0  [SS1 -> X20TB32v.SS; SL -> X20BM12w.SL1]
  Supervision = off
X20DO6639b : X20DO6639 v1.0.1.0  [SS1 -> X20TB32w.SS; SL -> X20BM12x.SL1]
  Supervision = off
X20DO6639c : X20DO6639 v1.0.1.0  [SS1 -> X20TB32x.SS; SL -> X20BM12y.SL1]
  Supervision = off
X20DO6639d : X20DO6639 v1.0.1.0  [SS1 -> X20TB32y.SS; SL -> X20BM12z.SL1]
  Supervision = off
X20DO6639e : X20DO6639 v1.0.1.0  [SS1 -> X20TB32z.SS; SL -> X20BM12aa.SL1]
  Supervision = off
X20DO6639f : X20DO6639 v1.0.1.0  [SS1 -> X20TB32aa.SS; SL -> X20BM12ab.SL1]
  Supervision = off
X20DO6639g : X20DO6639 v1.0.1.0  [SS1 -> X20TB32ab.SS; SL -> X20BM12ac.SL1]
  Supervision = off
X20DO6639h : X20DO6639 v1.0.1.0  [SS1 -> X20TB32ac.SS; SL -> X20BM12ad.SL1]
  Supervision = off
X20DO6639i : X20DO6639 v1.0.1.0  [SS1 -> X20TB32ad.SS; SL -> X20BM12ae.SL1]
  Supervision = off
X20DO6639j : X20DO6639 v1.0.1.0  [SS1 -> X20TB32ae.SS; SL -> X20BM12af.SL1]
  Supervision = off
X20DO6639k : X20DO6639 v1.0.1.0  [SS1 -> X20TB32af.SS; SL -> X20BM12ag.SL1]
  Supervision = off
X20DO6639l : X20DO6639 v1.0.1.0  [SS1 -> X20TB32ag.SS; SL -> X20BM12ah.SL1]
  Supervision = off
X20DO6639m : X20DO6639 v1.0.1.0  [SS1 -> X20TB32ah.SS; SL -> X20BM12ai.SL1]
  Supervision = off
X20PS3300 : X20PS3300 v1.1.0.0  [SS1 -> X20TB12g.SS; SL -> X20BM01.SL1]
  Supervision = off
X20PS3300a : X20PS3300 v1.1.0.0  [SS1 -> X20TB12f.SS; SL -> X20cBM01.SL1]
  Supervision = off
X20TB12 : X20TB12 v1.0.0.0
X20TB12a : X20TB12 v1.0.0.0
X20TB12b : X20TB12 v1.0.0.0
X20TB12c : X20TB12 v1.0.0.0
X20TB12d : X20TB12 v1.0.0.0
X20TB12e : X20TB12 v1.0.0.0
X20TB12f : X20TB12 v1.0.0.0
X20TB12g : X20TB12 v1.0.0.0
X20TB32 : X20TB32 v1.0.0.1
X20TB32a : X20TB32 v1.0.0.1
X20TB32aa : X20TB32 v1.0.0.1
X20TB32ab : X20TB32 v1.0.0.1
X20TB32ac : X20TB32 v1.0.0.1
X20TB32ad : X20TB32 v1.0.0.1
X20TB32ae : X20TB32 v1.0.0.1
X20TB32af : X20TB32 v1.0.0.1
X20TB32ag : X20TB32 v1.0.0.1
X20TB32ah : X20TB32 v1.0.0.1
X20TB32b : X20TB32 v1.0.0.1
X20TB32c : X20TB32 v1.0.0.1
X20TB32d : X20TB32 v1.0.0.1
X20TB32e : X20TB32 v1.0.0.1
X20TB32f : X20TB32 v1.0.0.1
X20TB32g : X20TB32 v1.0.0.1
X20TB32h : X20TB32 v1.0.0.1
X20TB32i : X20TB32 v1.0.0.1
X20TB32j : X20TB32 v1.0.0.1
X20TB32k : X20TB32 v1.0.0.1
X20TB32l : X20TB32 v1.0.0.1
X20TB32m : X20TB32 v1.0.0.1
X20TB32n : X20TB32 v1.0.0.1
X20TB32o : X20TB32 v1.0.0.1
X20TB32p : X20TB32 v1.0.0.1
X20TB32q : X20TB32 v1.0.0.1
X20TB32r : X20TB32 v1.0.0.1
X20TB32s : X20TB32 v1.0.0.1
X20TB32t : X20TB32 v1.0.0.1
X20TB32u : X20TB32 v1.0.0.1
X20TB32v : X20TB32 v1.0.0.1
X20TB32w : X20TB32 v1.0.0.1
X20TB32x : X20TB32 v1.0.0.1
X20TB32y : X20TB32 v1.0.0.1
X20TB32z : X20TB32 v1.0.0.1
X20cBM01 : X20cBM01 v1.0.1.0  [X2X1 -> X20BM12u.X2X2]
```

### Cpu.per - X20CP1584/Cpu.per
```iecst
VAR_CONFIG
	MarkEncoder AT %MD0; (* *)
END_VAR
```

### IoMap.iom - X20CP1584/IoMap.iom
```iecst
VAR_CONFIG
	Cyclic#1.ActlMetalEncoder AT %ID."X20DC137A".Encoder01;
	Cyclic#1.ActualDAC1 AT %QW."X20CM8281".AnalogOutput01;
	Cyclic#2.AmberLight AT %QX."X20DO6639".DigitalOutput02;
	Cyclic#2.BatchActivePhysical AT %QX."X20DO6639".DigitalOutput06;
	Cyclic#2.::BrakeEncoderReset AT %QX."X20DC137A3".Encoder01Reset;
	Cyclic#2.BlockingValve AT %QX."X20DO6639".DigitalOutput05;
	Cyclic#2.BlueLight AT %QX."X20DO6639".DigitalOutput03;
	Cyclic#2.BrakeArmLwrInhibit AT %IX."X20DI4653p".DigitalInput02;
	Cyclic#2.BrakeAutoIndicator AT %QX."X20DO6639l".DigitalOutput05;
	Cyclic#2.BrakeAutoRequest AT %IX."X20DI4653s".DigitalInput02;
	Cyclic#2.BrakeBeamDownProx AT %IX."X20DI4653q".DigitalInput02;
	Cyclic#2.BrakeBeamLower AT %QX."X20DO6639l".DigitalOutput02;
	Cyclic#2.BrakeBeamLwrInhibit AT %IX."X20DI4653p".DigitalInput03;
	Cyclic#2.BrakeBeamRaise AT %QX."X20DO6639l".DigitalOutput01;
	Cyclic#2.BrakeBeamUpProx AT %IX."X20DI4653q".DigitalInput03;
	Cyclic#2.BrakeCarriageJogIn AT %IX."X20DI4653s".DigitalInput03;
	Cyclic#2.BrakeCarriageJogOut AT %IX."X20DI4653s".DigitalInput04;
	Cyclic#2.BrakeEncoder AT %ID."X20DC137A3".Encoder01;
	Cyclic#2.BrakeHighSpeedRelay AT %QX."X20DO6639k".DigitalOutput03;
	Cyclic#2.BrakeHydraulics AT %IX."X20DI4653r".DigitalInput03;
	Cyclic#2.BrakeLeafHomeProx AT %IX."X20DI4653q".DigitalInput01;
	Cyclic#2.BrakeLeafLower AT %QX."X20DO6639l".DigitalOutput04;
	Cyclic#2.BrakeLeafRaise AT %QX."X20DO6639l".DigitalOutput03;
	Cyclic#2.BrakeManual AT %IX."X20DI4653s".DigitalInput01;
	Cyclic#2.BrakeOn AT %QX."X20DO6639m".DigitalOutput01;
	Cyclic#2.BrakePartPresent AT %IX."X20DI4653r".DigitalInput01;
	Cyclic#2.BrakeSequenceReset AT %IX."X20DI4653t".DigitalInput01;
	Cyclic#2.BrakeSetButton AT %IX."X20DI4653t".DigitalInput02;
	Cyclic#2.BrakeSingleCycle AT %IX."X20DI4653t".DigitalInput03;
	BrakeSpeedSwitch AT %IX."X20DI4653r".DigitalInput04;
	Cyclic#2.CarriageArmLower AT %QX."X20DO6639k".DigitalOutput05;
	Cyclic#2.CarriageArmRaise AT %QX."X20DO6639k".DigitalOutput04;
	Cyclic#2.CarriageClampClose AT %QX."X20DO6639k".DigitalOutput06;
	Cyclic#2.CarriageReference AT %IX."X20DI4653p".DigitalInput01;
	Cyclic#2.CenterShuttleOutput AT %QX."X20DO6639b".DigitalOutput01;
	Cyclic#2.CHoleValve AT %QX."X20DO6639b".DigitalOutput02;
	Cyclic#2.CleatRollerSheetSense AT %IX."X20DI4653j".DigitalInput03;
	Cyclic#2.DuctoAuto AT %IX."X20DI4653a".DigitalInput01;
	Cyclic#2.DuctSelected AT %IX."X20DI4653e".DigitalInput01;
	Cyclic#2.EjectComplete AT %IX."X20DI4653p".DigitalInput04;
	Cyclic#1.ElectricDriveEnable AT %QX."X20CM8281".DigitalOutput01;
	Cyclic#2.EStopClear AT %IX."X20DI4653".DigitalInput01;
	Cyclic#2.ExitBeltsOn AT %IX."X20DI4653j".DigitalInput01;
	Cyclic#2.FeedInitButton AT %IX."X20DI4653".DigitalInput04;
	Cyclic#2.InsulmaticEntranceHiSpeed AT %QX."X20DO6639m".DigitalOutput04;
	Cyclic#2.InsulmaticEntranceLowSpeed AT %QX."X20DO6639i".DigitalOutput02;
	Cyclic#2.GlueFlushPB AT %IX."X20DI4653l".DigitalInput03;
	Cyclic#2.GluePartSense AT %IX."X20DI4653l".DigitalInput02;
	Cyclic#2.GluePumpOnSwitch AT %IX."X20DI4653l".DigitalInput01;
	Cyclic#2.GlueServiceSwitch AT %IX."X20DI4653m".DigitalInput01;
	Cyclic#2.HumpLimitSwitch AT %IX."X20DI4653c".DigitalInput01;
	Cyclic#2.ImaticBladeDown AT %QX."X20DO6639j".DigitalOutput01;
	Cyclic#2.ImaticBladeUp AT %QX."X20DO6639i".DigitalOutput06;
	Cyclic#2.ImaticFeedRoll AT %QX."X20DO6639i".DigitalOutput03;
	Cyclic#2.ImaticPressRoll AT %QX."X20DO6639i".DigitalOutput04;
	Cyclic#2.::ISquarePinOn AT %IX."X20DI4653n".DigitalInput04;
	Cyclic#2.ImaticSquarePin AT %QX."X20DO6639i".DigitalOutput05;
	Cyclic#2.InsulationFeed AT %IX."X20DI4653n".DigitalInput03;
	Cyclic#2.InsulmaticExitHiSpeed AT %QX."X20DO6639m".DigitalOutput02;
	Cyclic#2.InsulmaticExitLowSpeed AT %QX."X20DO6639m".DigitalOutput03;
	Cyclic#2.InsulmaticOn AT %IX."X20DI4653n".DigitalInput01;
	LBrakePartEjectSolenoid AT %QX."X20DO6639l".DigitalOutput06;
	Cyclic#2.LeftShuttleOutput AT %QX."X20DO6639b".DigitalOutput03;
	Cyclic#2.LHoleValve AT %QX."X20DO6639b".DigitalOutput04;
	Cyclic#2.LTValve AT %QX."X20DO6639a".DigitalOutput04;
	Cyclic#2.MarkAuto AT %IX."X20DI4653d".DigitalInput02;
	Cyclic#2.MarkConveyorDelayFwd AT %IX."X20DI4653i".DigitalInput04;
	Cyclic#2.MarkEncoderResetSignal AT %QX."X20DC137A1".Encoder01Reset;
	Cyclic#2.MarkGateRaise AT %QX."X20DO6639f".DigitalOutput01;
	Cyclic#2.MarkHeadJogInSwitch AT %IX."X20DI4653e".DigitalInput03;
	Cyclic#2.MarkHeadJogOutSwitch AT %IX."X20DI4653e".DigitalInput04;
	Cyclic#2.MarkHiSpeedSignal AT %IX."X20DI4653e".DigitalInput02;
	Cyclic#2.MarkPshrFwd AT %QX."X20DO6639e".DigitalOutput06;
	Cyclic#2.MarkPushComplete AT %IX."X20DI4653h".DigitalInput02;
	Cyclic#2.MarkPusherStop AT %IX."X20DI4653i".DigitalInput01;
	Cyclic#2.MarkRefSwitch AT %IX."X20DI4653f".DigitalInput01;
	Cyclic#2.MarkRFHighSpeed AT %QX."X20DO6639c".DigitalOutput05;
	Cyclic#2.MarkRFMoveIn AT %QX."X20DO6639c".DigitalOutput03;
	Cyclic#2.MarkRFMoveOut AT %QX."X20DO6639c".DigitalOutput04;
	Cyclic#2.MarkRollformerOn AT %IX."X20DI4653d".DigitalInput01;
	Cyclic#2.MarkSetButton AT %IX."X20DI4653d".DigitalInput03;
	Cyclic#2.MarkTableFwd AT %QX."X20DO6639e".DigitalOutput03;
	Cyclic#2.::MarkTableStart AT %IX."X20DI4653g".DigitalInput01;
	Cyclic#2.MarkTableRev AT %QX."X20DO6639e".DigitalOutput04;
	Cyclic#2.MaterialClamped AT %IX."X20DI4653r".DigitalInput02;
	Cyclic#2.MatlAtMarkTable AT %IX."X20DI4653g".DigitalInput03;
	Cyclic#2.MatlAtMeasureRoll AT %IX."X20DI4653a".DigitalInput04;
	Cyclic#2.MoveAwayBeam AT %QX."X20DO6639k".DigitalOutput02;
	Cyclic#2.MoveToBeam AT %QX."X20DO6639k".DigitalOutput01;
	Cyclic#2.MTBlockedValve AT %QX."X20DO6639g".DigitalOutput06;
	Cyclic#2.MTFlushTubeCloseSolenoid AT %QX."X20DO6639h".DigitalOutput01;
	Cyclic#2.MTFlushTubeOpenSolenoid AT %QX."X20DO6639h".DigitalOutput02;
	Cyclic#2.MTGlueValveSolenoid AT %QX."X20DO6639h".DigitalOutput03;
	Cyclic#2.MTPlungerValveSolenoid AT %QX."X20DO6639h".DigitalOutput05;
	Cyclic#2.MTWaterFlushSolenoid AT %QX."X20DO6639h".DigitalOutput04;
	Cyclic#2.MTWaterSupplySolenoid AT %QX."X20DO6639h".DigitalOutput06;
	Cyclic#2.::LeftKnockDownRoll AT %QX."X20DO6639f".DigitalOutput03;
	Cyclic#2.PartAtInsulationFeed AT %IX."X20DI4653o".DigitalInput02;
	Cyclic#2.PartAtISquarePin AT %IX."X20DI4653o".DigitalInput01;
	Cyclic#2.PartPresentPSpotter AT %IX."X20DI4653o".DigitalInput03;
	Cyclic#2.PinspotEncoder AT %ID."X20DC137A2".Encoder01;
	Cyclic#2.PinspotEncoderResetSignal AT %QX."X20DC137A2".Encoder01Reset;
	Cyclic#2.PinspotterDrive AT %QX."X20DO6639j".DigitalOutput02;
	Cyclic#2.PinspotterLoad AT %QX."X20DO6639j".DigitalOutput03;
	Cyclic#2.PowerOn AT %IX."X20DI4653c".DigitalInput04;
	Cyclic#2.ProcessorDriveEnable AT %IX."X20DI4653".DigitalInput03;
	Cyclic#2.ProcessorJogFwd AT %IX."X20DI4653a".DigitalInput02;
	Cyclic#2.ProcessorJogRev AT %IX."X20DI4653a".DigitalInput03;
	Cyclic#2.RaiseImaticBlade AT %IX."X20DI4653n".DigitalInput02;
	Cyclic#2.RawMarkEncoder AT %ID."X20DC137A1".Encoder01;
	Cyclic#2.RHoleValve AT %QX."X20DO6639a".DigitalOutput06;
	Cyclic#2.RightShuttleOutput AT %QX."X20DO6639a".DigitalOutput05;
	Cyclic#2.ShearClampDownProx AT %IX."X20DI4653b".DigitalInput01;
	Cyclic#2.ShearClampLowerSolenoid AT %QX."X20DO6639b".DigitalOutput05;
	Cyclic#2.ShearClampRaiseSolenoid AT %QX."X20DO6639b".DigitalOutput06;
	Cyclic#2.ShearClampUpProx AT %IX."X20DI4653b".DigitalInput02;
	Cyclic#2.ShearLeafDownProx AT %IX."X20DI4653b".DigitalInput03;
	ShearLeafLowerSolenoid AT %QX."X20DO6639c".DigitalOutput01;
	ShearLeafRaiseSolenoid AT %QX."X20DO6639c".DigitalOutput02;
	Cyclic#2.ShearLeafUpProx AT %IX."X20DI4653b".DigitalInput04;
	Cyclic#2.ShearValve AT %QX."X20DO6639a".DigitalOutput01;
	Cyclic#2.SnapLockButtonGag AT %QX."X20DO6639a".DigitalOutput02;
	Cyclic#2.TDCPusherRevPB AT %IX."X20DI4653k".DigitalInput01;
	Cyclic#2.TDCPushPartPresent AT %IX."X20DI4653k".DigitalInput02;
	Cyclic#2.TDCPushStrokeComplete AT %IX."X20DI4653k".DigitalInput03;
	Cyclic#2.TDCRFPusherFwd AT %QX."X20DO6639g".DigitalOutput04;
	Cyclic#2.TDCRFPusherIndicator AT %IX."X20DI4653j".DigitalInput04;
	Cyclic#2.TDCRFPusherRev AT %QX."X20DO6639g".DigitalOutput05;
	Cyclic#2.TDCTablePartProx AT %IX."X20DI4653j".DigitalInput02;
	Cyclic#2.TDCTablePusherFwd AT %QX."X20DO6639f".DigitalOutput05;
	Cyclic#2.UncoilerRun AT %QX."X20DO6639".DigitalOutput04;
	Cyclic#2.VValve AT %QX."X20DO6639a".DigitalOutput03;
	Cyclic#2.WarningHorn AT %QX."X20DO6639".DigitalOutput01;
	Cyclic#2.WBrakeArmsUp AT %IX."X20DI4653q".DigitalInput04;
	Cyclic#2.UncoilerOnLatch AT %IX."X20DI4653".DigitalInput02;
	Cyclic#2.SlackBar AT %IX."X20DI4653c".DigitalInput02;
	Cyclic#2.UncoilerJogForwardPB AT %IX."X20DI4653h".DigitalInput03;
	Cyclic#2.UncoilerJogReversePB AT %IX."X20DI4653h".DigitalInput04;
	Cyclic#2.UncoilerForwardSolenoid AT %QX."X20DO6639d".DigitalOutput03;
	Cyclic#2.UncoilerReverseSolenoid AT %QX."X20DO6639d".DigitalOutput04;
	ShearBeamUpSS AT %IX."X20DI4653f".DigitalInput03;
	Cyclic#2.ShearBeamDownSS AT %IX."X20DI4653g".DigitalInput04;
	Cyclic#2.ShearLeafUpSS AT %IX."X20DI4653i".DigitalInput02;
	Cyclic#2.ShearLeafDownSS AT %IX."X20DI4653i".DigitalInput03;
	Cyclic#2.SystemHydraulicsOn AT %IX."X20DI4653k".DigitalInput04;
	Cyclic#2.::OneInchHolePunch AT %QX."X20DO6639f".DigitalOutput02;
	Cyclic#2.::RightKnockDownRoll AT %QX."X20DO6639f".DigitalOutput04;
	Cyclic#1.::ProcessorEncoderReset AT %QX."X20DC137A".Encoder01Reset;
	Cyclic#2.::GlueSprayEnable AT %QX."X20DO6639j".DigitalOutput04;
	Cyclic#2.::BrakeConveyorLow AT %QX."X20DO6639j".DigitalOutput05;
	Cyclic#2.::BrakeConveyorHigh AT %QX."X20DO6639j".DigitalOutput06;
END_VAR
```

## Configuration DUCTO2_V1

### Task classes (Cpu.sw)
```
Cyclic#1 (cycle 1000 us, tolerance 10000 us):
  IMotionCon <- IMotionControl.prg
  IMotion1 <- IMotion1.prg
  CleatRoll <- CleatRoll.prg
Cyclic#2 (cycle 10000 us, tolerance 20000 us):
  Uncoiler_1 <- Uncoiler_1.prg
  MarkTable <- MarkTable.prg
  MarkRF <- MarkRF.prg
  Feeder <- Feeder.prg
  SBrake <- SBrake.prg
  TDCTable <- TDCTable.prg
  TDCRFPshrs <- TDCRFPshrs.prg
  GlueApp <- GlueApp.prg
  Insulmatic <- Insulmatic.prg
  Pinspotter <- Pinspotter.prg
  BrakeCommo <- BrakeCommon.prg
  HydraulicB <- HydraulicBrakeCarriage.prg
  HWBwoPLC <- HWBwoPLC.prg
Cyclic#4 (cycle 100000 us, tolerance 100000 us):
  HMIButtons <- HMIButtons.prg
  Server <- LibAsTCP1_ST.Server.prg
Binaries: TCData, sysconf, Role, User, iomap, ashwd, asfw, arconfig
Libraries: standard, MestekLib, AsTCP, runtime, asstring, asieccon, astime
```

### Hardware
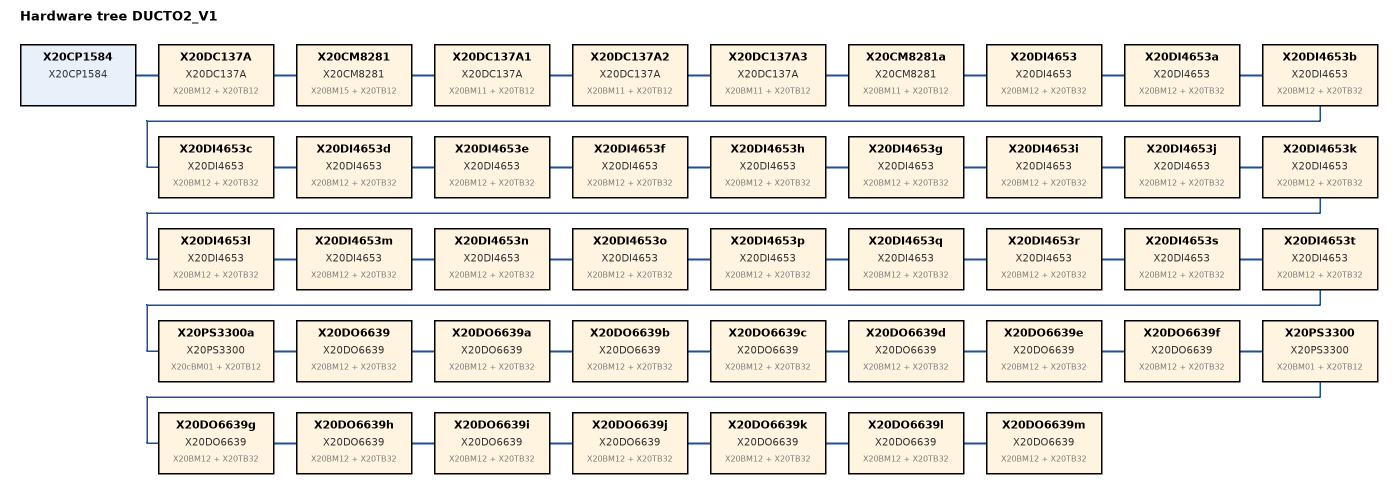
```
X20BM01 : X20BM01 v1.0.1.1  [X2X1 -> X20BM12ab.X2X2]
X20BM11a : X20BM11 v1.0.0.1  [X2X1 -> X20BM11b.X2X2]
X20BM11b : X20BM11 v1.0.0.1  [X2X1 -> X20BM15.X2X2]
X20BM11c : X20BM11 v1.0.0.1  [X2X1 -> X20BM11a.X2X2]
X20BM11d : X20BM11 v1.0.0.1  [X2X1 -> X20BM11c.X2X2]
X20BM12 : X20BM12 v1.0.0.1  [X2X1 -> X20BM11d.X2X2]
X20BM12a : X20BM12 v1.0.0.1  [X2X1 -> X20CP1584.IF6]
X20BM12aa : X20BM12 v1.0.0.1  [X2X1 -> X20BM12z.X2X2]
X20BM12ab : X20BM12 v1.0.0.1  [X2X1 -> X20BM12aa.X2X2]
X20BM12ac : X20BM12 v1.0.0.1  [X2X1 -> X20BM01.X2X2]
X20BM12ad : X20BM12 v1.0.0.1  [X2X1 -> X20BM12ac.X2X2]
X20BM12ae : X20BM12 v1.0.0.1  [X2X1 -> X20BM12ad.X2X2]
X20BM12af : X20BM12 v1.0.0.1  [X2X1 -> X20BM12ae.X2X2]
X20BM12ag : X20BM12 v1.0.0.1  [X2X1 -> X20BM12af.X2X2]
X20BM12ah : X20BM12 v1.0.0.1  [X2X1 -> X20BM12ag.X2X2]
X20BM12ai : X20BM12 v1.0.0.1  [X2X1 -> X20BM12ah.X2X2]
X20BM12b : X20BM12 v1.0.0.1  [X2X1 -> X20BM12.X2X2]
X20BM12c : X20BM12 v1.0.0.1  [X2X1 -> X20BM12b.X2X2]
X20BM12d : X20BM12 v1.0.0.1  [X2X1 -> X20BM12c.X2X2]
X20BM12e : X20BM12 v1.0.0.1  [X2X1 -> X20BM12d.X2X2]
X20BM12f : X20BM12 v1.0.0.1  [X2X1 -> X20BM12e.X2X2]
X20BM12g : X20BM12 v1.0.0.1  [X2X1 -> X20BM12f.X2X2]
X20BM12h : X20BM12 v1.0.0.1  [X2X1 -> X20BM12i.X2X2]
X20BM12i : X20BM12 v1.0.0.1  [X2X1 -> X20BM12g.X2X2]
X20BM12j : X20BM12 v1.0.0.1  [X2X1 -> X20BM12h.X2X2]
X20BM12k : X20BM12 v1.0.0.1  [X2X1 -> X20BM12j.X2X2]
X20BM12l : X20BM12 v1.0.0.1  [X2X1 -> X20BM12k.X2X2]
X20BM12m : X20BM12 v1.0.0.1  [X2X1 -> X20BM12l.X2X2]
X20BM12n : X20BM12 v1.0.0.1  [X2X1 -> X20BM12m.X2X2]
X20BM12o : X20BM12 v1.0.0.1  [X2X1 -> X20BM12n.X2X2]
X20BM12p : X20BM12 v1.0.0.1  [X2X1 -> X20BM12o.X2X2]
X20BM12q : X20BM12 v1.0.0.1  [X2X1 -> X20BM12p.X2X2]
X20BM12r : X20BM12 v1.0.0.1  [X2X1 -> X20BM12q.X2X2]
X20BM12s : X20BM12 v1.0.0.1  [X2X1 -> X20BM12r.X2X2]
X20BM12t : X20BM12 v1.0.0.1  [X2X1 -> X20BM12s.X2X2]
X20BM12u : X20BM12 v1.0.0.1  [X2X1 -> X20BM12t.X2X2]
X20BM12v : X20BM12 v1.0.0.1  [X2X1 -> X20cBM01.X2X2]
X20BM12w : X20BM12 v1.0.0.1  [X2X1 -> X20BM12v.X2X2]
X20BM12x : X20BM12 v1.0.0.1  [X2X1 -> X20BM12w.X2X2]
X20BM12y : X20BM12 v1.0.0.1  [X2X1 -> X20BM12x.X2X2]
X20BM12z : X20BM12 v1.0.0.1  [X2X1 -> X20BM12y.X2X2]
X20BM15 : X20BM15 v1.0.1.0  [X2X1 -> X20BM12a.X2X2 (NodeNumber=2)]
X20CM8281 : X20CM8281 v1.0.4.0  [SS1 -> X20TB12.SS; SL -> X20BM15.SL1]
  Supervision = off
X20CM8281a : X20CM8281 v1.0.4.0  [SS1 -> X20TB12e.SS; SL -> X20BM11d.SL1]
  Supervision = off
X20CP1584 : X20CP1584 v1.3.0.0
  Connector IF2:
    ActivateDevice = 1
    EthInterfaceRedundant = 0
    Mode = Manual
    InternetAddress = 10.1.254.101
  Connector IF3:
    EplInterfaceRedundant = 0
    EplEthInterfaceRedundant = 0
  ConfigurationID = X20_CPU_test
  EnableUsbRemoteInstall = 1
  TimerDeviceType = SWIOTIMER
  Cyclic1Duration = 1000
  Cyclic1Tolerance = 10000
  Cyclic2Duration = 10000
  Cyclic2Tolerance = 20000
  Cyclic3Duration = 50000
  Cyclic3Tolerance = 50000
  Cyclic4Duration = 100000
  Cyclic4Tolerance = 100000
  Cyclic5Duration = 200000
  Cyclic5Tolerance = 200000
  Cyclic6Duration = 500000
  Cyclic6Tolerance = 500000
  Cyclic7Duration = 1000000
  Cyclic7Tolerance = 1000000
  Cyclic8Duration = 10000
  Cyclic8Tolerance = 30000000
X20DC137A : X20DC137A v1.0.0.3 (LastFrozenVersion=1.0.0.3)  [SS1 -> X20TB12b.SS; SL -> X20BM12a.SL1]
  Supervision = off
  CounterStd01 = 32Bit
  BWConfigChannel03 = off
X20DC137A1 : X20DC137A v1.0.0.3 (LastFrozenVersion=1.0.0.3)  [SS1 -> X20TB12c.SS; SL -> X20BM11b.SL1]
  Supervision = off
  CounterStd01 = 32Bit
  BWConfigChannel03 = off
X20DC137A2 : X20DC137A v1.0.0.3 (LastFrozenVersion=1.0.0.3)  [SS1 -> X20TB12a.SS; SL -> X20BM11a.SL1]
  Supervision = off
  CounterStd01 = 32Bit
  BWConfigChannel03 = off
X20DC137A3 : X20DC137A v1.0.0.3 (LastFrozenVersion=1.0.0.3)  [SS1 -> X20TB12d.SS; SL -> X20BM11c.SL1]
  Supervision = off
  CounterStd01 = 32Bit
  BWConfigChannel03 = off
X20DI4653 : X20DI4653 v1.0.2.0  [SS1 -> X20TB32.SS; SL -> X20BM12.SL1]
  Supervision = off
X20DI4653a : X20DI4653 v1.0.2.0  [SS1 -> X20TB32a.SS; SL -> X20BM12b.SL1]
  Supervision = off
X20DI4653b : X20DI4653 v1.0.2.0  [SS1 -> X20TB32b.SS; SL -> X20BM12c.SL1]
  Supervision = off
X20DI4653c : X20DI4653 v1.0.2.0  [SS1 -> X20TB32c.SS; SL -> X20BM12d.SL1]
  Supervision = off
X20DI4653d : X20DI4653 v1.0.2.0  [SS1 -> X20TB32d.SS; SL -> X20BM12e.SL1]
  Supervision = off
X20DI4653e : X20DI4653 v1.0.2.0  [SS1 -> X20TB32e.SS; SL -> X20BM12f.SL1]
  Supervision = off
X20DI4653f : X20DI4653 v1.0.2.0  [SS1 -> X20TB32f.SS; SL -> X20BM12g.SL1]
  Supervision = off
X20DI4653g : X20DI4653 v1.0.2.0  [SS1 -> X20TB32g.SS; SL -> X20BM12h.SL1]
  Supervision = off
X20DI4653h : X20DI4653 v1.0.2.0  [SS1 -> X20TB32h.SS; SL -> X20BM12i.SL1]
  Supervision = off
X20DI4653i : X20DI4653 v1.0.2.0  [SS1 -> X20TB32i.SS; SL -> X20BM12j.SL1]
  Supervision = off
X20DI4653j : X20DI4653 v1.0.2.0  [SS1 -> X20TB32j.SS; SL -> X20BM12k.SL1]
  Supervision = off
X20DI4653k : X20DI4653 v1.0.2.0  [SS1 -> X20TB32k.SS; SL -> X20BM12l.SL1]
  Supervision = off
X20DI4653l : X20DI4653 v1.0.2.0  [SS1 -> X20TB32l.SS; SL -> X20BM12m.SL1]
  Supervision = off
X20DI4653m : X20DI4653 v1.0.2.0  [SS1 -> X20TB32m.SS; SL -> X20BM12n.SL1]
  Supervision = off
X20DI4653n : X20DI4653 v1.0.2.0  [SS1 -> X20TB32n.SS; SL -> X20BM12o.SL1]
  Supervision = off
X20DI4653o : X20DI4653 v1.0.2.0  [SS1 -> X20TB32o.SS; SL -> X20BM12p.SL1]
  Supervision = off
X20DI4653p : X20DI4653 v1.0.2.0  [SS1 -> X20TB32p.SS; SL -> X20BM12q.SL1]
  Supervision = off
X20DI4653q : X20DI4653 v1.0.2.0  [SS1 -> X20TB32q.SS; SL -> X20BM12r.SL1]
  Supervision = off
X20DI4653r : X20DI4653 v1.0.2.0  [SS1 -> X20TB32r.SS; SL -> X20BM12s.SL1]
  Supervision = off
X20DI4653s : X20DI4653 v1.0.2.0  [SS1 -> X20TB32s.SS; SL -> X20BM12t.SL1]
  Supervision = off
X20DI4653t : X20DI4653 v1.0.2.0  [SS1 -> X20TB32t.SS; SL -> X20BM12u.SL1]
  Supervision = off
X20DO6639 : X20DO6639 v1.0.1.0  [SS1 -> X20TB32u.SS; SL -> X20BM12v.SL1]
  Supervision = off
X20DO6639a : X20DO6639 v1.0.1.0  [SS1 -> X20TB32v.SS; SL -> X20BM12w.SL1]
  Supervision = off
X20DO6639b : X20DO6639 v1.0.1.0  [SS1 -> X20TB32w.SS; SL -> X20BM12x.SL1]
  Supervision = off
X20DO6639c : X20DO6639 v1.0.1.0  [SS1 -> X20TB32x.SS; SL -> X20BM12y.SL1]
  Supervision = off
X20DO6639d : X20DO6639 v1.0.1.0  [SS1 -> X20TB32y.SS; SL -> X20BM12z.SL1]
  Supervision = off
X20DO6639e : X20DO6639 v1.0.1.0  [SS1 -> X20TB32z.SS; SL -> X20BM12aa.SL1]
  Supervision = off
X20DO6639f : X20DO6639 v1.0.1.0  [SS1 -> X20TB32aa.SS; SL -> X20BM12ab.SL1]
  Supervision = off
X20DO6639g : X20DO6639 v1.0.1.0  [SS1 -> X20TB32ab.SS; SL -> X20BM12ac.SL1]
  Supervision = off
X20DO6639h : X20DO6639 v1.0.1.0  [SS1 -> X20TB32ac.SS; SL -> X20BM12ad.SL1]
  Supervision = off
X20DO6639i : X20DO6639 v1.0.1.0  [SS1 -> X20TB32ad.SS; SL -> X20BM12ae.SL1]
  Supervision = off
X20DO6639j : X20DO6639 v1.0.1.0  [SS1 -> X20TB32ae.SS; SL -> X20BM12af.SL1]
  Supervision = off
X20DO6639k : X20DO6639 v1.0.1.0  [SS1 -> X20TB32af.SS; SL -> X20BM12ag.SL1]
  Supervision = off
X20DO6639l : X20DO6639 v1.0.1.0  [SS1 -> X20TB32ag.SS; SL -> X20BM12ah.SL1]
  Supervision = off
X20DO6639m : X20DO6639 v1.0.1.0  [SS1 -> X20TB32ah.SS; SL -> X20BM12ai.SL1]
  Supervision = off
X20PS3300 : X20PS3300 v1.1.0.0  [SS1 -> X20TB12g.SS; SL -> X20BM01.SL1]
  Supervision = off
X20PS3300a : X20PS3300 v1.1.0.0  [SS1 -> X20TB12f.SS; SL -> X20cBM01.SL1]
  Supervision = off
X20TB12 : X20TB12 v1.0.0.0
X20TB12a : X20TB12 v1.0.0.0
X20TB12b : X20TB12 v1.0.0.0
X20TB12c : X20TB12 v1.0.0.0
X20TB12d : X20TB12 v1.0.0.0
X20TB12e : X20TB12 v1.0.0.0
X20TB12f : X20TB12 v1.0.0.0
X20TB12g : X20TB12 v1.0.0.0
X20TB32 : X20TB32 v1.0.0.1
X20TB32a : X20TB32 v1.0.0.1
X20TB32aa : X20TB32 v1.0.0.1
X20TB32ab : X20TB32 v1.0.0.1
X20TB32ac : X20TB32 v1.0.0.1
X20TB32ad : X20TB32 v1.0.0.1
X20TB32ae : X20TB32 v1.0.0.1
X20TB32af : X20TB32 v1.0.0.1
X20TB32ag : X20TB32 v1.0.0.1
X20TB32ah : X20TB32 v1.0.0.1
X20TB32b : X20TB32 v1.0.0.1
X20TB32c : X20TB32 v1.0.0.1
X20TB32d : X20TB32 v1.0.0.1
X20TB32e : X20TB32 v1.0.0.1
X20TB32f : X20TB32 v1.0.0.1
X20TB32g : X20TB32 v1.0.0.1
X20TB32h : X20TB32 v1.0.0.1
X20TB32i : X20TB32 v1.0.0.1
X20TB32j : X20TB32 v1.0.0.1
X20TB32k : X20TB32 v1.0.0.1
X20TB32l : X20TB32 v1.0.0.1
X20TB32m : X20TB32 v1.0.0.1
X20TB32n : X20TB32 v1.0.0.1
X20TB32o : X20TB32 v1.0.0.1
X20TB32p : X20TB32 v1.0.0.1
X20TB32q : X20TB32 v1.0.0.1
X20TB32r : X20TB32 v1.0.0.1
X20TB32s : X20TB32 v1.0.0.1
X20TB32t : X20TB32 v1.0.0.1
X20TB32u : X20TB32 v1.0.0.1
X20TB32v : X20TB32 v1.0.0.1
X20TB32w : X20TB32 v1.0.0.1
X20TB32x : X20TB32 v1.0.0.1
X20TB32y : X20TB32 v1.0.0.1
X20TB32z : X20TB32 v1.0.0.1
X20cBM01 : X20cBM01 v1.0.1.0  [X2X1 -> X20BM12u.X2X2]
```

### IoMap.iom - X20CP1584/IoMap.iom
```iecst
VAR_CONFIG
	Cyclic#1.ActlMetalEncoder AT %ID."X20DC137A".Encoder01;
	Cyclic#1.::ProcessorEncoderReset AT %QX."X20DC137A".Encoder01Reset;
	Cyclic#1.ActualDAC1 AT %QW."X20CM8281".AnalogOutput01;
	Cyclic#1.ElectricDriveEnable AT %QX."X20CM8281".DigitalOutput01;
	Cyclic#2.MarkEncoderResetSignal AT %QX."X20DC137A1".Encoder01Reset;
	Cyclic#2.RawMarkEncoder AT %ID."X20DC137A1".Encoder01;
	Cyclic#2.PinspotEncoder AT %ID."X20DC137A2".Encoder01;
	Cyclic#2.PinspotEncoderResetSignal AT %QX."X20DC137A2".Encoder01Reset;
	Cyclic#2.::BrakeEncoderReset AT %QX."X20DC137A3".Encoder01Reset;
	Cyclic#2.BrakeEncoder AT %ID."X20DC137A3".Encoder01;
	Cyclic#2.EStopClear AT %IX."X20DI4653".DigitalInput01;
	Cyclic#2.FeedInitButton AT %IX."X20DI4653".DigitalInput04;
	Cyclic#2.ProcessorDriveEnable AT %IX."X20DI4653".DigitalInput03;
	Cyclic#2.UncoilerOnLatch AT %IX."X20DI4653".DigitalInput02;
	Cyclic#2.DuctoAuto AT %IX."X20DI4653a".DigitalInput01;
	Cyclic#2.MatlAtMeasureRoll AT %IX."X20DI4653a".DigitalInput04;
	Cyclic#2.ProcessorJogFwd AT %IX."X20DI4653a".DigitalInput02;
	Cyclic#2.ProcessorJogRev AT %IX."X20DI4653a".DigitalInput03;
	Cyclic#2.ShearClampDownProx AT %IX."X20DI4653b".DigitalInput01;
	Cyclic#2.ShearClampUpProx AT %IX."X20DI4653b".DigitalInput02;
	Cyclic#2.ShearLeafDownProx AT %IX."X20DI4653b".DigitalInput03;
	Cyclic#2.ShearLeafUpProx AT %IX."X20DI4653b".DigitalInput04;
	Cyclic#2.HumpLimitSwitch AT %IX."X20DI4653c".DigitalInput01;
	Cyclic#2.PowerOn AT %IX."X20DI4653c".DigitalInput04;
	Cyclic#2.SlackBar AT %IX."X20DI4653c".DigitalInput02;
	::PartPresentMarkExit AT %IX."X20DI4653c".DigitalInput03;
	Cyclic#2.MarkAuto AT %IX."X20DI4653d".DigitalInput02;
	Cyclic#2.MarkRollformerOn AT %IX."X20DI4653d".DigitalInput01;
	Cyclic#2.MarkSetButton AT %IX."X20DI4653d".DigitalInput03;
	Cyclic#2.SmallPittsSelected AT %IX."X20DI4653d".DigitalInput04;
	Cyclic#2.DuctSelected AT %IX."X20DI4653e".DigitalInput01;
	Cyclic#2.MarkHeadJogInSwitch AT %IX."X20DI4653e".DigitalInput03;
	Cyclic#2.MarkHeadJogOutSwitch AT %IX."X20DI4653e".DigitalInput04;
	Cyclic#2.MarkHiSpeedSignal AT %IX."X20DI4653e".DigitalInput02;
	Cyclic#2.MarkRefSwitch AT %IX."X20DI4653f".DigitalInput01;
	Cyclic#2.ShearBeamUpSS AT %IX."X20DI4653f".DigitalInput03;
	Cyclic#2.MarkPushComplete AT %IX."X20DI4653h".DigitalInput02;
	Cyclic#2.::Mark3PusherHome AT %IX."X20DI4653h".DigitalInput03;
	Cyclic#2.UncoilerJogReversePB AT %IX."X20DI4653h".DigitalInput04;
	Cyclic#2.::MarkTableStart AT %IX."X20DI4653g".DigitalInput01;
	Cyclic#2.MatlAtMarkTable AT %IX."X20DI4653g".DigitalInput03;
	Cyclic#2.ShearBeamDownSS AT %IX."X20DI4653g".DigitalInput04;
	Cyclic#2.::MarkTTPusherJogRevPB AT %IX."X20DI4653g".DigitalInput02;
	Cyclic#2.MarkConveyorDelayFwd AT %IX."X20DI4653i".DigitalInput04;
	Cyclic#2.MarkPusherStop AT %IX."X20DI4653i".DigitalInput01;
	Cyclic#2.ShearLeafUpSS AT %IX."X20DI4653i".DigitalInput02;
	Cyclic#2.ShearLeafDownSS AT %IX."X20DI4653i".DigitalInput03;
	Cyclic#2.CleatRollerSheetSense AT %IX."X20DI4653j".DigitalInput03;
	Cyclic#2.ExitBeltsOn AT %IX."X20DI4653j".DigitalInput01;
	Cyclic#2.::TDCRFPusherStart AT %IX."X20DI4653j".DigitalInput04;
	Cyclic#2.TDCTablePartProx AT %IX."X20DI4653j".DigitalInput02;
	Cyclic#2.TDCPusherRevPB AT %IX."X20DI4653k".DigitalInput01;
	Cyclic#2.TDCPushPartPresent AT %IX."X20DI4653k".DigitalInput02;
	Cyclic#2.TDCPushStrokeComplete AT %IX."X20DI4653k".DigitalInput03;
	Cyclic#2.SystemHydraulicsOn AT %IX."X20DI4653k".DigitalInput04;
	Cyclic#2.GlueFlushPB AT %IX."X20DI4653l".DigitalInput03;
	Cyclic#2.GluePartSense AT %IX."X20DI4653l".DigitalInput02;
	Cyclic#2.GluePumpOnSwitch AT %IX."X20DI4653l".DigitalInput01;
	Cyclic#2.::InsulmaticOnA AT %IX."X20DI4653l".DigitalInput04;
	Cyclic#2.GlueServiceSwitch AT %IX."X20DI4653m".DigitalInput01;
	Cyclic#2.::ISquarePinOn AT %IX."X20DI4653n".DigitalInput04;
	Cyclic#2.InsulationFeed AT %IX."X20DI4653n".DigitalInput03;
	Cyclic#2.RaiseImaticBlade AT %IX."X20DI4653n".DigitalInput02;
	Cyclic#2.InsulmaticOnB AT %IX."X20DI4653n".DigitalInput01;
	Cyclic#2.::PartAtInsulationFeed AT %IX."X20DI4653o".DigitalInput02;
	Cyclic#2.::PartAtISquarePin AT %IX."X20DI4653o".DigitalInput01;
	Cyclic#2.::BrakeActive AT %IX."X20DI4653o".DigitalInput04;
	Cyclic#2.::PartPresentPSpotter AT %IX."X20DI4653o".DigitalInput03;
	Cyclic#2.BrakeArmLwrInhibit AT %IX."X20DI4653p".DigitalInput02;
	Cyclic#2.BrakeBeamLwrInhibit AT %IX."X20DI4653p".DigitalInput03;
	Cyclic#2.CarriageReference AT %IX."X20DI4653p".DigitalInput01;
	Cyclic#2.EjectComplete AT %IX."X20DI4653p".DigitalInput04;
	Cyclic#2.BrakeBeamDownProx AT %IX."X20DI4653q".DigitalInput02;
	Cyclic#2.BrakeBeamUpProx AT %IX."X20DI4653q".DigitalInput03;
	Cyclic#2.BrakeLeafHomeProx AT %IX."X20DI4653q".DigitalInput01;
	Cyclic#2.diWBrakeArmsUp AT %IX."X20DI4653q".DigitalInput04;
	Cyclic#2.BrakeHydraulics AT %IX."X20DI4653r".DigitalInput03;
	Cyclic#2.BrakePartPresent AT %IX."X20DI4653r".DigitalInput01;
	Cyclic#2.BrakeSpeedSwitch AT %IX."X20DI4653r".DigitalInput04;
	Cyclic#2.MaterialClamped AT %IX."X20DI4653r".DigitalInput02;
	Cyclic#2.BrakeAutoRequest AT %IX."X20DI4653s".DigitalInput02;
	Cyclic#2.diBrakeCarriageJogIn AT %IX."X20DI4653s".DigitalInput03;
	Cyclic#2.diBrakeCarriageJogOut AT %IX."X20DI4653s".DigitalInput04;
	Cyclic#2.BrakeManualButton AT %IX."X20DI4653s".DigitalInput01;
	Cyclic#2.BrakeSequenceReset AT %IX."X20DI4653t".DigitalInput01;
	Cyclic#2.BrakeSetButton AT %IX."X20DI4653t".DigitalInput02;
	Cyclic#2.BrakeSingleCycle AT %IX."X20DI4653t".DigitalInput03;
	Cyclic#2.::BendInProcess AT %IX."X20DI4653t".DigitalInput04;
	Cyclic#2.AmberLight AT %QX."X20DO6639".DigitalOutput02;
	Cyclic#2.BatchActivePhysical AT %QX."X20DO6639".DigitalOutput06;
	Cyclic#2.BlockingValve AT %QX."X20DO6639".DigitalOutput05;
	Cyclic#2.BlueLight AT %QX."X20DO6639".DigitalOutput03;
	Cyclic#2.UncoilerRun AT %QX."X20DO6639".DigitalOutput04;
	Cyclic#2.WarningHorn AT %QX."X20DO6639".DigitalOutput01;
	Cyclic#2.LTValve AT %QX."X20DO6639a".DigitalOutput04;
	Cyclic#2.RHoleValve AT %QX."X20DO6639a".DigitalOutput06;
	Cyclic#2.RightShuttleOutput AT %QX."X20DO6639a".DigitalOutput05;
	Cyclic#2.ShearValve AT %QX."X20DO6639a".DigitalOutput01;
	Cyclic#2.SnapLockButtonGag AT %QX."X20DO6639a".DigitalOutput02;
	Cyclic#2.VValve AT %QX."X20DO6639a".DigitalOutput03;
	Cyclic#2.CenterShuttleOutput AT %QX."X20DO6639b".DigitalOutput01;
	Cyclic#2.CHoleValve AT %QX."X20DO6639b".DigitalOutput02;
	Cyclic#2.LeftShuttleOutput AT %QX."X20DO6639b".DigitalOutput03;
	Cyclic#2.LHoleValve AT %QX."X20DO6639b".DigitalOutput04;
	Cyclic#2.ShearClampLowerSolenoid AT %QX."X20DO6639b".DigitalOutput05;
	Cyclic#2.ShearClampRaiseSolenoid AT %QX."X20DO6639b".DigitalOutput06;
	Cyclic#2.MarkRFHighSpeed AT %QX."X20DO6639c".DigitalOutput05;
	Cyclic#2.MarkRFMoveIn AT %QX."X20DO6639c".DigitalOutput03;
	Cyclic#2.MarkRFMoveOut AT %QX."X20DO6639c".DigitalOutput04;
	ShearLeafLowerSolenoid AT %QX."X20DO6639c".DigitalOutput01;
	ShearLeafRaiseSolenoid AT %QX."X20DO6639c".DigitalOutput02;
	Cyclic#2.UncoilerForwardSolenoid AT %QX."X20DO6639d".DigitalOutput03;
	Cyclic#2.UncoilerReverseSolenoid AT %QX."X20DO6639d".DigitalOutput04;
	Cyclic#2.MarkPusherReverse AT %QX."X20DO6639d".DigitalOutput01;
	Cyclic#2.MarkPshrFwd AT %QX."X20DO6639e".DigitalOutput06;
	Cyclic#2.MarkTableFwd AT %QX."X20DO6639e".DigitalOutput03;
	Cyclic#2.MarkTableRev AT %QX."X20DO6639e".DigitalOutput04;
	Cyclic#2.MarkGateRaise AT %QX."X20DO6639f".DigitalOutput01;
	Cyclic#2.::LeftKnockDownRoll AT %QX."X20DO6639f".DigitalOutput03;
	Cyclic#2.TDCTablePusherFwd AT %QX."X20DO6639f".DigitalOutput05;
	Cyclic#2.::OneInchHolePunch AT %QX."X20DO6639f".DigitalOutput02;
	Cyclic#2.::RightKnockDownRoll AT %QX."X20DO6639f".DigitalOutput04;
	Cyclic#2.MTBlockedValve AT %QX."X20DO6639g".DigitalOutput06;
	Cyclic#2.TDCRFPusherFwd AT %QX."X20DO6639g".DigitalOutput04;
	Cyclic#2.TDCRFPusherRev AT %QX."X20DO6639g".DigitalOutput05;
	Cyclic#2.MTFlushTubeCloseSolenoid AT %QX."X20DO6639h".DigitalOutput01;
	Cyclic#2.MTFlushTubeOpenSolenoid AT %QX."X20DO6639h".DigitalOutput02;
	Cyclic#2.MTGlueValveSolenoid AT %QX."X20DO6639h".DigitalOutput03;
	Cyclic#2.MTPlungerValveSolenoid AT %QX."X20DO6639h".DigitalOutput05;
	Cyclic#2.MTWaterFlushSolenoid AT %QX."X20DO6639h".DigitalOutput04;
	Cyclic#2.MTWaterSupplySolenoid AT %QX."X20DO6639h".DigitalOutput06;
	Cyclic#2.InsulmaticEntranceLowSpeed AT %QX."X20DO6639i".DigitalOutput02;
	Cyclic#2.ImaticBladeUp AT %QX."X20DO6639i".DigitalOutput06;
	Cyclic#2.ImaticFeedRoll AT %QX."X20DO6639i".DigitalOutput03;
	Cyclic#2.ImaticPressRoll AT %QX."X20DO6639i".DigitalOutput04;
	Cyclic#2.ImaticSquarePin AT %QX."X20DO6639i".DigitalOutput05;
	Cyclic#2.ImaticBladeDown AT %QX."X20DO6639j".DigitalOutput01;
	Cyclic#2.PinspotterDrive AT %QX."X20DO6639j".DigitalOutput02;
	Cyclic#2.PinspotterLoad AT %QX."X20DO6639j".DigitalOutput03;
	Cyclic#2.::GlueSprayEnable AT %QX."X20DO6639j".DigitalOutput04;
	Cyclic#2.::BrakeConveyorLow AT %QX."X20DO6639j".DigitalOutput05;
	Cyclic#2.::BrakeConveyorHigh AT %QX."X20DO6639j".DigitalOutput06;
	Cyclic#2.BrakeHighSpeedRelay AT %QX."X20DO6639k".DigitalOutput03;
	Cyclic#2.CarriageArmLower AT %QX."X20DO6639k".DigitalOutput05;
	Cyclic#2.CarriageArmRaise AT %QX."X20DO6639k".DigitalOutput04;
	Cyclic#2.CarriageClampClose AT %QX."X20DO6639k".DigitalOutput06;
	Cyclic#2.MoveAwayBeam AT %QX."X20DO6639k".DigitalOutput02;
	Cyclic#2.MoveToBeam AT %QX."X20DO6639k".DigitalOutput01;
	Cyclic#2.BrakeAutoIndicator AT %QX."X20DO6639l".DigitalOutput05;
	Cyclic#2.BrakeBeamLower AT %QX."X20DO6639l".DigitalOutput02;
	Cyclic#2.BrakeBeamRaise AT %QX."X20DO6639l".DigitalOutput01;
	Cyclic#2.BrakeLeafLower AT %QX."X20DO6639l".DigitalOutput04;
	Cyclic#2.BrakeLeafRaise AT %QX."X20DO6639l".DigitalOutput03;
	Cyclic#2.LBrakePartEjectSolenoid AT %QX."X20DO6639l".DigitalOutput06;
	Cyclic#2.BrakeOn AT %QX."X20DO6639m".DigitalOutput01;
	Cyclic#2.InsulmaticEntranceHiSpeed AT %QX."X20DO6639m".DigitalOutput04;
	Cyclic#2.InsulmaticExitHiSpeed AT %QX."X20DO6639m".DigitalOutput02;
	Cyclic#2.InsulmaticExitLowSpeed AT %QX."X20DO6639m".DigitalOutput03;
	Cyclic#2.::BendStart AT %QX."X20DO6639m".DigitalOutput05;
	Cyclic#2.SealantValve AT %QX."X20DO6639d".DigitalOutput02;
	Cyclic#2.::doMarkRollformerHeadRaise AT %QX."X20DO6639d".DigitalOutput05;
	Cyclic#2.::doMarkRollformerHeadLower AT %QX."X20DO6639d".DigitalOutput06;
	Cyclic#2.::doMarkRFPassUp AT %QX."X20DO6639e".DigitalOutput01;
	Cyclic#2.::doMarkRFPassUp AT %QX."X20DO6639e".DigitalOutput02;
	Cyclic#2.::doTDCAdjustableHeadIn AT %QX."X20DO6639f".DigitalOutput06;
	Cyclic#2.::doTDCAdjustableHeadOut AT %QX."X20DO6639g".DigitalOutput01;
	Cyclic#2.::doTDCFixedHeadIn AT %QX."X20DO6639g".DigitalOutput02;
	Cyclic#2.::doTDCFixedHeadOut AT %QX."X20DO6639g".DigitalOutput03;
	Cyclic#1.::BrakeDriveEnable AT %QX."X20CM8281a".DigitalOutput01;
	::ActualDAC2 AT %QW."X20CM8281a".AnalogOutput01;
	Cyclic#1.BrakeDriveFaultReset AT %QX."X20CM8281a".DigitalOutput02;
	Cyclic#1.::BrakeDriveReady AT %IX."X20CM8281a".DigitalInput01;
	::diMarkHeadUpProx AT %IX."X20DI4653f".DigitalInput04;
	::diMarkHeadDownProx AT %IX."X20DI4653h".DigitalInput01;
END_VAR
```

### OpcArMap.opcc - X20CP1584/OpcArMap.opcc
```
Map:
  Tag MakeBeadRollTable (Scope=)
    PV MakeBeadRollTable (Task=, DataType=boolean, IsVector=False, BitNumber=none)
  Tag MakeButtonTable (Scope=)
    PV MakeButtonTable (Task=, DataType=boolean, IsVector=False, BitNumber=none)
  Tag MakeCHoleTable (Scope=)
    PV MakeCHoleTable (Task=, DataType=boolean, IsVector=False, BitNumber=none)
  Tag MakeCleatTable (Scope=)
    PV MakeCleatTable (Task=, DataType=boolean, IsVector=False, BitNumber=none)
  Tag MakeCustomLTTable (Scope=)
    PV MakeCustomLTTable (Task=, DataType=boolean, IsVector=False, BitNumber=none)
  Tag MakeCustomVTable (Scope=)
    PV MakeCustomVTable (Task=, DataType=boolean, IsVector=False, BitNumber=none)
  Tag MakeLHoleTable (Scope=)
    PV MakeLHoleTable (Task=, DataType=boolean, IsVector=False, BitNumber=none)
  Tag MakeLTTable (Scope=)
    PV MakeLTTable (Task=, DataType=boolean, IsVector=False, BitNumber=none)
  Tag MakeRHoleTable (Scope=)
    PV MakeRHoleTable (Task=, DataType=boolean, IsVector=False, BitNumber=none)
  Tag MakeShearBrakeTable (Scope=)
    PV MakeShearBrakeTable (Task=, DataType=boolean, IsVector=False, BitNumber=none)
  Tag MakeShearTable (Scope=)
    PV MakeShearTable (Task=, DataType=boolean, IsVector=False, BitNumber=none)
  Tag MakeVTable (Scope=)
    PV MakeVTable (Task=, DataType=boolean, IsVector=False, BitNumber=none)
```

## Configuration DUCTO2_V2

### Task classes (Cpu.sw)
```
Cyclic#1 (cycle 1000 us, tolerance 10000 us):
  EMotionCon <- EMotionControl.prg
Cyclic#2 (cycle 20000 us, tolerance 20000 us):
  MarkTable <- MarkTable.prg
  MarkRF <- MarkRF.prg
  Feeder <- Feeder.prg
  TDCTable <- TDCTable.prg
  TDCRFPshrs <- TDCRFPshrs.prg
  GlueApp <- GlueApp.prg
  Insulmatic <- Insulmatic.prg
  Pinspotter <- Pinspotter.prg
  BrakeCommo <- BrakeCommon.prg
  HydraulicB <- HydraulicBrakeCarriage.prg
  HWBwoPLC <- HWBwoPLC.prg
  CleatRoll <- CleatRoll.prg
Cyclic#4 (cycle 100000 us, tolerance 100000 us):
  HMIButtons <- HMIButtons.prg
  Server <- LibAsTCP1_ST.Server.prg
Binaries: sysconf, Role, User, iomap, ashwd, asfw, arconfig, TCData
Libraries: standard, MestekLib, AsTCP, runtime, asstring, asieccon, astime
```

### Hardware
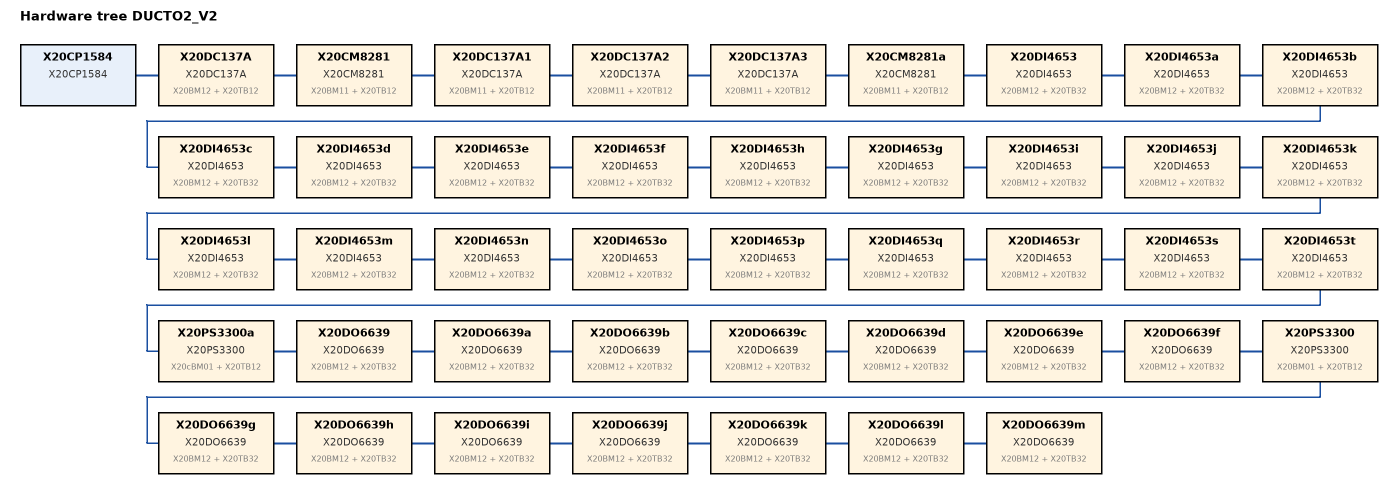
```
X20BM01 : X20BM01 v1.0.1.1  [X2X1 -> X20BM12ab.X2X2]
X20BM11 : X20BM11 v1.0.0.1  [X2X1 -> X20BM12a.X2X2]
X20BM11a : X20BM11 v1.0.0.1  [X2X1 -> X20BM11b.X2X2]
X20BM11b : X20BM11 v1.0.0.1  [X2X1 -> X20BM11.X2X2]
X20BM11c : X20BM11 v1.0.0.1  [X2X1 -> X20BM11a.X2X2]
X20BM11d : X20BM11 v1.0.0.1  [X2X1 -> X20BM11c.X2X2]
X20BM12 : X20BM12 v1.0.0.1  [X2X1 -> X20BM11d.X2X2]
X20BM12a : X20BM12 v1.0.0.1  [X2X1 -> X20CP1584.IF6]
X20BM12aa : X20BM12 v1.0.0.1  [X2X1 -> X20BM12z.X2X2]
X20BM12ab : X20BM12 v1.0.0.1  [X2X1 -> X20BM12aa.X2X2]
X20BM12ac : X20BM12 v1.0.0.1  [X2X1 -> X20BM01.X2X2]
X20BM12ad : X20BM12 v1.0.0.1  [X2X1 -> X20BM12ac.X2X2]
X20BM12ae : X20BM12 v1.0.0.1  [X2X1 -> X20BM12ad.X2X2]
X20BM12af : X20BM12 v1.0.0.1  [X2X1 -> X20BM12ae.X2X2]
X20BM12ag : X20BM12 v1.0.0.1  [X2X1 -> X20BM12af.X2X2]
X20BM12ah : X20BM12 v1.0.0.1  [X2X1 -> X20BM12ag.X2X2]
X20BM12ai : X20BM12 v1.0.0.1  [X2X1 -> X20BM12ah.X2X2]
X20BM12b : X20BM12 v1.0.0.1  [X2X1 -> X20BM12.X2X2]
X20BM12c : X20BM12 v1.0.0.1  [X2X1 -> X20BM12b.X2X2]
X20BM12d : X20BM12 v1.0.0.1  [X2X1 -> X20BM12c.X2X2]
X20BM12e : X20BM12 v1.0.0.1  [X2X1 -> X20BM12d.X2X2]
X20BM12f : X20BM12 v1.0.0.1  [X2X1 -> X20BM12e.X2X2]
X20BM12g : X20BM12 v1.0.0.1  [X2X1 -> X20BM12f.X2X2]
X20BM12h : X20BM12 v1.0.0.1  [X2X1 -> X20BM12i.X2X2]
X20BM12i : X20BM12 v1.0.0.1  [X2X1 -> X20BM12g.X2X2]
X20BM12j : X20BM12 v1.0.0.1  [X2X1 -> X20BM12h.X2X2]
X20BM12k : X20BM12 v1.0.0.1  [X2X1 -> X20BM12j.X2X2]
X20BM12l : X20BM12 v1.0.0.1  [X2X1 -> X20BM12k.X2X2]
X20BM12m : X20BM12 v1.0.0.1  [X2X1 -> X20BM12l.X2X2]
X20BM12n : X20BM12 v1.0.0.1  [X2X1 -> X20BM12m.X2X2]
X20BM12o : X20BM12 v1.0.0.1  [X2X1 -> X20BM12n.X2X2]
X20BM12p : X20BM12 v1.0.0.1  [X2X1 -> X20BM12o.X2X2]
X20BM12q : X20BM12 v1.0.0.1  [X2X1 -> X20BM12p.X2X2]
X20BM12r : X20BM12 v1.0.0.1  [X2X1 -> X20BM12q.X2X2]
X20BM12s : X20BM12 v1.0.0.1  [X2X1 -> X20BM12r.X2X2]
X20BM12t : X20BM12 v1.0.0.1  [X2X1 -> X20BM12s.X2X2]
X20BM12u : X20BM12 v1.0.0.1  [X2X1 -> X20BM12t.X2X2]
X20BM12v : X20BM12 v1.0.0.1  [X2X1 -> X20cBM01.X2X2]
X20BM12w : X20BM12 v1.0.0.1  [X2X1 -> X20BM12v.X2X2]
X20BM12x : X20BM12 v1.0.0.1  [X2X1 -> X20BM12w.X2X2]
X20BM12y : X20BM12 v1.0.0.1  [X2X1 -> X20BM12x.X2X2]
X20BM12z : X20BM12 v1.0.0.1  [X2X1 -> X20BM12y.X2X2]
X20CM8281 : X20CM8281 v1.0.4.0  [SS1 -> X20TB12.SS; SL -> X20BM11.SL1]
  Supervision = off
X20CM8281a : X20CM8281 v1.0.4.0  [SS1 -> X20TB12e.SS; SL -> X20BM11d.SL1]
  Supervision = off
X20CP1584 : X20CP1584 v1.3.0.0
  Connector IF2:
    ActivateDevice = 1
    EthInterfaceRedundant = 0
    Mode = Manual
    InternetAddress = 10.1.254.101
  Connector IF3:
    EplInterfaceRedundant = 0
    EplEthInterfaceRedundant = 0
  ConfigurationID = X20_CPU_test
  EnableUsbRemoteInstall = 1
  TimerDeviceType = SWIOTIMER
  Cyclic1Duration = 1000
  Cyclic1Tolerance = 10000
  Cyclic2Duration = 20000
  Cyclic2Tolerance = 20000
  Cyclic3Duration = 50000
  Cyclic3Tolerance = 50000
  Cyclic4Duration = 100000
  Cyclic4Tolerance = 100000
  Cyclic5Duration = 200000
  Cyclic5Tolerance = 200000
  Cyclic6Duration = 500000
  Cyclic6Tolerance = 500000
  Cyclic7Duration = 1000000
  Cyclic7Tolerance = 1000000
  Cyclic8Duration = 10000
  Cyclic8Tolerance = 30000000
X20DC137A : X20DC137A v1.0.0.3  [SS1 -> X20TB12b.SS; SL -> X20BM12a.SL1]
  Supervision = off
  CounterStd01 = 32Bit
  BWConfigChannel03 = off
X20DC137A1 : X20DC137A v1.0.0.3  [SS1 -> X20TB12c.SS; SL -> X20BM11b.SL1]
  Supervision = off
  CounterStd01 = 32Bit
  BWConfigChannel03 = off
X20DC137A2 : X20DC137A v1.0.0.3  [SS1 -> X20TB12a.SS; SL -> X20BM11a.SL1]
  Supervision = off
  CounterStd01 = 32Bit
  BWConfigChannel03 = off
X20DC137A3 : X20DC137A v1.0.0.3  [SS1 -> X20TB12d.SS; SL -> X20BM11c.SL1]
  Supervision = off
  CounterStd01 = 32Bit
  BWConfigChannel03 = off
X20DI4653 : X20DI4653 v1.0.2.0  [SS1 -> X20TB32.SS; SL -> X20BM12.SL1]
  Supervision = off
X20DI4653a : X20DI4653 v1.0.2.0  [SS1 -> X20TB32a.SS; SL -> X20BM12b.SL1]
  Supervision = off
X20DI4653b : X20DI4653 v1.0.2.0  [SS1 -> X20TB32b.SS; SL -> X20BM12c.SL1]
  Supervision = off
X20DI4653c : X20DI4653 v1.0.2.0  [SS1 -> X20TB32c.SS; SL -> X20BM12d.SL1]
  Supervision = off
X20DI4653d : X20DI4653 v1.0.2.0  [SS1 -> X20TB32d.SS; SL -> X20BM12e.SL1]
  Supervision = off
X20DI4653e : X20DI4653 v1.0.2.0  [SS1 -> X20TB32e.SS; SL -> X20BM12f.SL1]
  Supervision = off
X20DI4653f : X20DI4653 v1.0.2.0  [SS1 -> X20TB32f.SS; SL -> X20BM12g.SL1]
  Supervision = off
X20DI4653g : X20DI4653 v1.0.2.0  [SS1 -> X20TB32g.SS; SL -> X20BM12h.SL1]
  Supervision = off
X20DI4653h : X20DI4653 v1.0.2.0  [SS1 -> X20TB32h.SS; SL -> X20BM12i.SL1]
  Supervision = off
X20DI4653i : X20DI4653 v1.0.2.0  [SS1 -> X20TB32i.SS; SL -> X20BM12j.SL1]
  Supervision = off
X20DI4653j : X20DI4653 v1.0.2.0  [SS1 -> X20TB32j.SS; SL -> X20BM12k.SL1]
  Supervision = off
X20DI4653k : X20DI4653 v1.0.2.0  [SS1 -> X20TB32k.SS; SL -> X20BM12l.SL1]
  Supervision = off
X20DI4653l : X20DI4653 v1.0.2.0  [SS1 -> X20TB32l.SS; SL -> X20BM12m.SL1]
  Supervision = off
X20DI4653m : X20DI4653 v1.0.2.0  [SS1 -> X20TB32m.SS; SL -> X20BM12n.SL1]
  Supervision = off
X20DI4653n : X20DI4653 v1.0.2.0  [SS1 -> X20TB32n.SS; SL -> X20BM12o.SL1]
  Supervision = off
X20DI4653o : X20DI4653 v1.0.2.0  [SS1 -> X20TB32o.SS; SL -> X20BM12p.SL1]
  Supervision = off
X20DI4653p : X20DI4653 v1.0.2.0  [SS1 -> X20TB32p.SS; SL -> X20BM12q.SL1]
  Supervision = off
X20DI4653q : X20DI4653 v1.0.2.0  [SS1 -> X20TB32q.SS; SL -> X20BM12r.SL1]
  Supervision = off
X20DI4653r : X20DI4653 v1.0.2.0  [SS1 -> X20TB32r.SS; SL -> X20BM12s.SL1]
  Supervision = off
X20DI4653s : X20DI4653 v1.0.2.0  [SS1 -> X20TB32s.SS; SL -> X20BM12t.SL1]
  Supervision = off
X20DI4653t : X20DI4653 v1.0.2.0  [SS1 -> X20TB32t.SS; SL -> X20BM12u.SL1]
  Supervision = off
X20DO6639 : X20DO6639 v1.0.1.0  [SS1 -> X20TB32u.SS; SL -> X20BM12v.SL1]
  Supervision = off
X20DO6639a : X20DO6639 v1.0.1.0  [SS1 -> X20TB32v.SS; SL -> X20BM12w.SL1]
  Supervision = off
X20DO6639b : X20DO6639 v1.0.1.0  [SS1 -> X20TB32w.SS; SL -> X20BM12x.SL1]
  Supervision = off
X20DO6639c : X20DO6639 v1.0.1.0  [SS1 -> X20TB32x.SS; SL -> X20BM12y.SL1]
  Supervision = off
X20DO6639d : X20DO6639 v1.0.1.0  [SS1 -> X20TB32y.SS; SL -> X20BM12z.SL1]
  Supervision = off
X20DO6639e : X20DO6639 v1.0.1.0  [SS1 -> X20TB32z.SS; SL -> X20BM12aa.SL1]
  Supervision = off
X20DO6639f : X20DO6639 v1.0.1.0  [SS1 -> X20TB32aa.SS; SL -> X20BM12ab.SL1]
  Supervision = off
X20DO6639g : X20DO6639 v1.0.1.0  [SS1 -> X20TB32ab.SS; SL -> X20BM12ac.SL1]
  Supervision = off
X20DO6639h : X20DO6639 v1.0.1.0  [SS1 -> X20TB32ac.SS; SL -> X20BM12ad.SL1]
  Supervision = off
X20DO6639i : X20DO6639 v1.0.1.0  [SS1 -> X20TB32ad.SS; SL -> X20BM12ae.SL1]
  Supervision = off
X20DO6639j : X20DO6639 v1.0.1.0  [SS1 -> X20TB32ae.SS; SL -> X20BM12af.SL1]
  Supervision = off
X20DO6639k : X20DO6639 v1.0.1.0  [SS1 -> X20TB32af.SS; SL -> X20BM12ag.SL1]
  Supervision = off
X20DO6639l : X20DO6639 v1.0.1.0  [SS1 -> X20TB32ag.SS; SL -> X20BM12ah.SL1]
  Supervision = off
X20DO6639m : X20DO6639 v1.0.1.0  [SS1 -> X20TB32ah.SS; SL -> X20BM12ai.SL1]
  Supervision = off
X20PS3300 : X20PS3300 v1.1.0.0  [SS1 -> X20TB12g.SS; SL -> X20BM01.SL1]
  Supervision = off
X20PS3300a : X20PS3300 v1.1.0.0  [SS1 -> X20TB12f.SS; SL -> X20cBM01.SL1]
  Supervision = off
X20TB12 : X20TB12 v1.0.0.0
X20TB12a : X20TB12 v1.0.0.0
X20TB12b : X20TB12 v1.0.0.0
X20TB12c : X20TB12 v1.0.0.0
X20TB12d : X20TB12 v1.0.0.0
X20TB12e : X20TB12 v1.0.0.0
X20TB12f : X20TB12 v1.0.0.0
X20TB12g : X20TB12 v1.0.0.0
X20TB32 : X20TB32 v1.0.0.1
X20TB32a : X20TB32 v1.0.0.1
X20TB32aa : X20TB32 v1.0.0.1
X20TB32ab : X20TB32 v1.0.0.1
X20TB32ac : X20TB32 v1.0.0.1
X20TB32ad : X20TB32 v1.0.0.1
X20TB32ae : X20TB32 v1.0.0.1
X20TB32af : X20TB32 v1.0.0.1
X20TB32ag : X20TB32 v1.0.0.1
X20TB32ah : X20TB32 v1.0.0.1
X20TB32b : X20TB32 v1.0.0.1
X20TB32c : X20TB32 v1.0.0.1
X20TB32d : X20TB32 v1.0.0.1
X20TB32e : X20TB32 v1.0.0.1
X20TB32f : X20TB32 v1.0.0.1
X20TB32g : X20TB32 v1.0.0.1
X20TB32h : X20TB32 v1.0.0.1
X20TB32i : X20TB32 v1.0.0.1
X20TB32j : X20TB32 v1.0.0.1
X20TB32k : X20TB32 v1.0.0.1
X20TB32l : X20TB32 v1.0.0.1
X20TB32m : X20TB32 v1.0.0.1
X20TB32n : X20TB32 v1.0.0.1
X20TB32o : X20TB32 v1.0.0.1
X20TB32p : X20TB32 v1.0.0.1
X20TB32q : X20TB32 v1.0.0.1
X20TB32r : X20TB32 v1.0.0.1
X20TB32s : X20TB32 v1.0.0.1
X20TB32t : X20TB32 v1.0.0.1
X20TB32u : X20TB32 v1.0.0.1
X20TB32v : X20TB32 v1.0.0.1
X20TB32w : X20TB32 v1.0.0.1
X20TB32x : X20TB32 v1.0.0.1
X20TB32y : X20TB32 v1.0.0.1
X20TB32z : X20TB32 v1.0.0.1
X20cBM01 : X20cBM01 v1.0.1.0  [X2X1 -> X20BM12u.X2X2]
```

### IoMap.iom - X20CP1584/IoMap.iom
```iecst
VAR_CONFIG
	Cyclic#1.ActlMetalEncoder AT %ID."X20DC137A".Encoder01;
	Cyclic#1.ActualDAC1 AT %QW."X20CM8281".AnalogOutput01;
	Cyclic#1.ElectricDriveEnable AT %QX."X20CM8281".DigitalOutput01;
	Cyclic#2.RawMarkEncoder AT %ID."X20DC137A1".Encoder01;
	Cyclic#2.PinspotEncoder AT %ID."X20DC137A2".Encoder01;
	Cyclic#2.BrakeEncoder AT %ID."X20DC137A3".Encoder01;
	Cyclic#2.EStopClear AT %IX."X20DI4653".DigitalInput01;
	Cyclic#2.FeedInitButton AT %IX."X20DI4653".DigitalInput04;
	Cyclic#2.ProcessorDriveEnable AT %IX."X20DI4653".DigitalInput03;
	Cyclic#2.DuctoAuto AT %IX."X20DI4653a".DigitalInput01;
	Cyclic#2.ProcessorJogFwd AT %IX."X20DI4653a".DigitalInput02;
	Cyclic#2.ProcessorJogRev AT %IX."X20DI4653a".DigitalInput03;
	Cyclic#2.MatlAtMeasureRoll AT %IX."X20DI4653a".DigitalInput04;
	::PowerOn AT %IX."X20DI4653c".DigitalInput04;
	Cyclic#2.MarkAuto AT %IX."X20DI4653d".DigitalInput02;
	Cyclic#2.MarkSetButton AT %IX."X20DI4653d".DigitalInput03;
	Cyclic#2.DuctSelected AT %IX."X20DI4653e".DigitalInput01;
	Cyclic#2.MarkHiSpeedSignal AT %IX."X20DI4653e".DigitalInput02;
	Cyclic#2.MarkHeadJogInSwitch AT %IX."X20DI4653e".DigitalInput03;
	Cyclic#2.MarkHeadJogOutSwitch AT %IX."X20DI4653e".DigitalInput04;
	Cyclic#2.MarkRefSwitch AT %IX."X20DI4653f".DigitalInput01;
	Cyclic#2.MarkPushComplete AT %IX."X20DI4653h".DigitalInput02;
	Cyclic#2.MarkTableOn AT %IX."X20DI4653g".DigitalInput01;
	Cyclic#2.MatlAtMarkTable AT %IX."X20DI4653g".DigitalInput03;
	Cyclic#2.MarkPusherStop AT %IX."X20DI4653i".DigitalInput01;
	Cyclic#2.MarkConveyorDelayFwd AT %IX."X20DI4653i".DigitalInput04;
	Cyclic#2.ExitBeltsOn AT %IX."X20DI4653j".DigitalInput01;
	Cyclic#2.CleatRollerSheetSense AT %IX."X20DI4653j".DigitalInput03;
	Cyclic#2.TDCRFPusherIndicator AT %IX."X20DI4653j".DigitalInput04;
	Cyclic#2.TDCPusherRevPB AT %IX."X20DI4653k".DigitalInput01;
	Cyclic#2.TDCPushPartPresent AT %IX."X20DI4653k".DigitalInput02;
	Cyclic#2.TDCPushStrokeComplete AT %IX."X20DI4653k".DigitalInput03;
	Cyclic#2.InsulmaticOn AT %IX."X20DI4653n".DigitalInput01;
	Cyclic#2.RaiseImaticBlade AT %IX."X20DI4653n".DigitalInput02;
	Cyclic#2.InsulationFeed AT %IX."X20DI4653n".DigitalInput03;
	Cyclic#2.ImaticSquarePin AT %IX."X20DI4653n".DigitalInput04;
	Cyclic#2.PartAtInsulationFeed AT %IX."X20DI4653o".DigitalInput01;
	Cyclic#2.PartAtISquarePin AT %IX."X20DI4653o".DigitalInput02;
	Cyclic#2.PartPresentPSpotter AT %IX."X20DI4653o".DigitalInput03;
	Cyclic#2.EjectComplete AT %IX."X20DI4653p".DigitalInput04;
	Cyclic#2.BrakeLeafHomeProx AT %IX."X20DI4653q".DigitalInput01;
	Cyclic#2.BrakeBeamDownProx AT %IX."X20DI4653q".DigitalInput02;
	Cyclic#2.BrakeBeamUpProx AT %IX."X20DI4653q".DigitalInput03;
	Cyclic#2.WBrakeArmsUp AT %IX."X20DI4653q".DigitalInput04;
	Cyclic#2.BrakePartPresent AT %IX."X20DI4653r".DigitalInput01;
	Cyclic#2.MaterialClamped AT %IX."X20DI4653r".DigitalInput02;
	Cyclic#2.BrakeHydraulics AT %IX."X20DI4653r".DigitalInput03;
	Cyclic#2.::BrakeAutoRequest AT %IX."X20DI4653s".DigitalInput02;
	Cyclic#2.BrakeCarriageJogIn AT %IX."X20DI4653s".DigitalInput03;
	Cyclic#2.BrakeCarriageJogOut AT %IX."X20DI4653s".DigitalInput04;
	Cyclic#2.BrakeSequenceReset AT %IX."X20DI4653t".DigitalInput01;
	Cyclic#2.BrakeSetButton AT %IX."X20DI4653t".DigitalInput02;
	Cyclic#2.BrakeSingleCycle AT %IX."X20DI4653t".DigitalInput03;
	Cyclic#2.WarningHorn AT %QX."X20DO6639".DigitalOutput01;
	Cyclic#2.AmberLight AT %QX."X20DO6639".DigitalOutput02;
	Cyclic#2.BlueLight AT %QX."X20DO6639".DigitalOutput03;
	Cyclic#2.UncoilerRun AT %QX."X20DO6639".DigitalOutput04;
	Cyclic#2.BlockingValve AT %QX."X20DO6639".DigitalOutput05;
	Cyclic#2.BatchActivePhysical AT %QX."X20DO6639".DigitalOutput06;
	Cyclic#2.ShearValve AT %QX."X20DO6639a".DigitalOutput01;
	Cyclic#2.SnapLockButtonGag AT %QX."X20DO6639a".DigitalOutput02;
	Cyclic#2.VValve AT %QX."X20DO6639a".DigitalOutput03;
	Cyclic#2.LTValve AT %QX."X20DO6639a".DigitalOutput04;
	Cyclic#2.RightShuttleOutput AT %QX."X20DO6639a".DigitalOutput05;
	Cyclic#2.RHoleValve AT %QX."X20DO6639a".DigitalOutput06;
	Cyclic#2.CenterShuttleOutput AT %QX."X20DO6639b".DigitalOutput01;
	Cyclic#2.CHoleValve AT %QX."X20DO6639b".DigitalOutput02;
	Cyclic#2.LeftShuttleOutput AT %QX."X20DO6639b".DigitalOutput03;
	Cyclic#2.LHoleValve AT %QX."X20DO6639b".DigitalOutput04;
	Cyclic#2.MarkRFMoveIn AT %QX."X20DO6639c".DigitalOutput03;
	Cyclic#2.MarkRFMoveOut AT %QX."X20DO6639c".DigitalOutput04;
	Cyclic#2.MarkRFHighSpeed AT %QX."X20DO6639c".DigitalOutput05;
	Cyclic#2.MarkTableFwd AT %QX."X20DO6639e".DigitalOutput03;
	Cyclic#2.MarkTableRev AT %QX."X20DO6639e".DigitalOutput04;
	Cyclic#2.MarkPshrFwd AT %QX."X20DO6639e".DigitalOutput06;
	Cyclic#2.MarkGateRaise AT %QX."X20DO6639f".DigitalOutput01;
	Cyclic#2.TDCTablePusherFwd AT %QX."X20DO6639f".DigitalOutput05;
	Cyclic#2.TDCRFPusherFwd AT %QX."X20DO6639g".DigitalOutput04;
	Cyclic#2.TDCRFPusherRev AT %QX."X20DO6639g".DigitalOutput05;
	Cyclic#2.ImaticFeedRoll AT %QX."X20DO6639i".DigitalOutput02;
	Cyclic#2.ImaticPressRoll AT %QX."X20DO6639i".DigitalOutput03;
	Cyclic#2.ImaticSquarePin AT %QX."X20DO6639i".DigitalOutput04;
	Cyclic#2.ImaticBladeUp AT %QX."X20DO6639i".DigitalOutput05;
	Cyclic#2.ImaticBladeDown AT %QX."X20DO6639j".DigitalOutput01;
	Cyclic#2.PinspotterDrive AT %QX."X20DO6639j".DigitalOutput02;
	Cyclic#2.PinspotterLoad AT %QX."X20DO6639j".DigitalOutput03;
	Cyclic#2.MoveToBeam AT %QX."X20DO6639k".DigitalOutput01;
	Cyclic#2.MoveAwayBeam AT %QX."X20DO6639k".DigitalOutput02;
	Cyclic#2.BrakeHighSpeedRelay AT %QX."X20DO6639k".DigitalOutput03;
	Cyclic#2.CarriageArmRaise AT %QX."X20DO6639k".DigitalOutput04;
	Cyclic#2.CarriageArmLower AT %QX."X20DO6639k".DigitalOutput05;
	Cyclic#2.CarriageClampClose AT %QX."X20DO6639k".DigitalOutput06;
	Cyclic#2.BrakeBeamRaise AT %QX."X20DO6639l".DigitalOutput01;
	Cyclic#2.BrakeOn AT %QX."X20DO6639m".DigitalOutput01;
	Cyclic#2.::CarriageReference AT %IX."X20DI4653p".DigitalInput01;
	Cyclic#2.::BrakeArmLwrInhibit AT %IX."X20DI4653p".DigitalInput02;
	Cyclic#2.::BrakeBeamLwrInhibit AT %IX."X20DI4653p".DigitalInput03;
	Cyclic#2.::BrakeBeamLower AT %QX."X20DO6639l".DigitalOutput02;
	Cyclic#2.::BrakeLeafRaise AT %QX."X20DO6639l".DigitalOutput03;
	Cyclic#2.::BrakeLeafLower AT %QX."X20DO6639l".DigitalOutput04;
	Cyclic#2.::BrakeAutoIndicator AT %QX."X20DO6639l".DigitalOutput05;
	Cyclic#2.BC_Home4 AT %QX."X20DC137A3".Encoder01Reset;
	BrakeSpeedSwitch AT %IX."X20DI4653r".DigitalInput04;
	BrakeManual AT %IX."X20DI4653s".DigitalInput01;
	LBrakePartEjectSolenoid AT %QX."X20DO6639l".DigitalOutput06;
	Cyclic#2.MarkEncoderResetSignal AT %QX."X20DC137A1".Encoder01Reset;
	Cyclic#2.::PinspotEncoderResetSignal AT %QX."X20DC137A2".Encoder01Reset;
END_VAR
```

## Configuration E1000

CPU X20CP1584, AutomationRuntime J4.25, Build 4.1.2, Vc V4.25.0

### Hardware
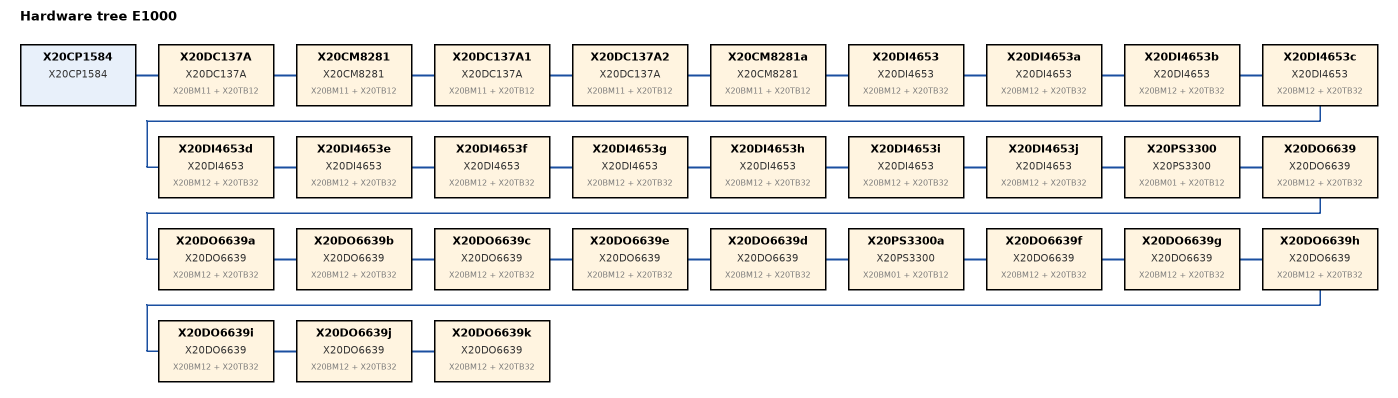
```
X20BM01 : X20BM01 v1.0.1.1  [X2X1 -> X20BM12j.X2X2]
X20BM01a : X20BM01 v1.0.1.1  [X2X1 -> X20BM12o.X2X2]
X20BM11 : X20BM11 v1.0.0.1  [X2X1 -> X20CP1584.IF6]
X20BM11a : X20BM11 v1.0.0.1  [X2X1 -> X20BM11.X2X2]
X20BM11b : X20BM11 v1.0.0.1  [X2X1 -> X20BM11a.X2X2]
X20BM11c : X20BM11 v1.0.0.1  [X2X1 -> X20BM11b.X2X2]
X20BM11d : X20BM11 v1.0.0.1  [X2X1 -> X20BM11c.X2X2]
X20BM12 : X20BM12 v1.0.0.1  [X2X1 -> X20BM11d.X2X2]
X20BM12a : X20BM12 v1.0.0.1  [X2X1 -> X20BM12.X2X2]
X20BM12b : X20BM12 v1.0.0.1  [X2X1 -> X20BM12a.X2X2]
X20BM12c : X20BM12 v1.0.0.1  [X2X1 -> X20BM12b.X2X2]
X20BM12d : X20BM12 v1.0.0.1  [X2X1 -> X20BM12c.X2X2]
X20BM12e : X20BM12 v1.0.0.1  [X2X1 -> X20BM12d.X2X2]
X20BM12f : X20BM12 v1.0.0.1  [X2X1 -> X20BM12e.X2X2]
X20BM12g : X20BM12 v1.0.0.1  [X2X1 -> X20BM12f.X2X2]
X20BM12h : X20BM12 v1.0.0.1  [X2X1 -> X20BM12g.X2X2]
X20BM12i : X20BM12 v1.0.0.1  [X2X1 -> X20BM12h.X2X2]
X20BM12j : X20BM12 v1.0.0.1  [X2X1 -> X20BM12i.X2X2]
X20BM12k : X20BM12 v1.0.0.1  [X2X1 -> X20BM01.X2X2]
X20BM12l : X20BM12 v1.0.0.1  [X2X1 -> X20BM12k.X2X2]
X20BM12m : X20BM12 v1.0.0.1  [X2X1 -> X20BM12l.X2X2]
X20BM12n : X20BM12 v1.0.0.1  [X2X1 -> X20BM12m.X2X2]
X20BM12o : X20BM12 v1.0.0.1  [X2X1 -> X20BM12p.X2X2]
X20BM12p : X20BM12 v1.0.0.1  [X2X1 -> X20BM12n.X2X2]
X20BM12q : X20BM12 v1.0.0.1  [X2X1 -> X20BM01a.X2X2]
X20BM12r : X20BM12 v1.0.0.1  [X2X1 -> X20BM12q.X2X2]
X20BM12s : X20BM12 v1.0.0.1  [X2X1 -> X20BM12r.X2X2]
X20BM12t : X20BM12 v1.0.0.1  [X2X1 -> X20BM12s.X2X2]
X20BM12u : X20BM12 v1.0.0.1  [X2X1 -> X20BM12t.X2X2]
X20BM12v : X20BM12 v1.0.0.1  [X2X1 -> X20BM12u.X2X2]
X20CM8281 : X20CM8281 v1.0.4.0  [SS1 -> X20TB12a.SS; SL -> X20BM11a.SL1]
  Supervision = off
X20CM8281a : X20CM8281 v1.0.4.0  [SS1 -> X20TB12d.SS; SL -> X20BM11d.SL1]
  Supervision = off
X20CP1584 : X20CP1584 v1.3.0.0
  Connector IF2:
    ActivateDevice = 1
    EthInterfaceRedundant = 0
    Mode = Manual
    InternetAddress = 10.1.254.101
  Connector IF3:
    EplInterfaceRedundant = 0
    EplEthInterfaceRedundant = 0
  Connector IF6:
    CycleTime = 1000
  ConfigurationID = X20_CPU_E1000
  EnableUsbRemoteInstall = 1
  TimerDeviceType = EPLX2X
  TimerDevice = X20CP1584.IF6
  Cyclic1Duration = 1000
  Cyclic1Tolerance = 0
  Cyclic1Output = 1
  Cyclic2Duration = 20000
  Cyclic2Tolerance = 20000
  Cyclic3Duration = 50000
  Cyclic3Tolerance = 50000
  Cyclic4Duration = 100000
  Cyclic4Tolerance = 100000
  Cyclic5Duration = 200000
  Cyclic5Tolerance = 200000
  Cyclic6Duration = 500000
  Cyclic6Tolerance = 500000
  Cyclic7Duration = 1000000
  Cyclic7Tolerance = 1000000
  Cyclic8Duration = 10000
  Cyclic8Tolerance = 30000000
  Route1
  DestinationAddress1 = 10.1.254.101
  SubnetMask1 = 255.0.0.0
X20DC137A : X20DC137A v1.0.0.3  [SS1 -> X20TB12.SS; SL -> X20BM11.SL1]
  Supervision = off
  CounterStd01 = 32Bit
  BWConfigChannel03 = off
X20DC137A1 : X20DC137A v1.0.0.3  [SS1 -> X20TB12b.SS; SL -> X20BM11b.SL1]
  Supervision = off
X20DC137A2 : X20DC137A v1.0.0.3  [SS1 -> X20TB12c.SS; SL -> X20BM11c.SL1]
  Supervision = off
X20DI4653 : X20DI4653 v1.0.2.0  [SS1 -> X20TB32.SS; SL -> X20BM12.SL1]
  Supervision = off
X20DI4653a : X20DI4653 v1.0.2.0  [SS1 -> X20TB32a.SS; SL -> X20BM12a.SL1]
  Supervision = off
X20DI4653b : X20DI4653 v1.0.2.0  [SS1 -> X20TB32b.SS; SL -> X20BM12b.SL1]
  Supervision = off
X20DI4653c : X20DI4653 v1.0.2.0  [SS1 -> X20TB32c.SS; SL -> X20BM12c.SL1]
  Supervision = off
X20DI4653d : X20DI4653 v1.0.2.0  [SS1 -> X20TB32d.SS; SL -> X20BM12d.SL1]
  Supervision = off
X20DI4653e : X20DI4653 v1.0.2.0  [SS1 -> X20TB32e.SS; SL -> X20BM12e.SL1]
  Supervision = off
X20DI4653f : X20DI4653 v1.0.2.0  [SS1 -> X20TB32f.SS; SL -> X20BM12f.SL1]
  Supervision = off
X20DI4653g : X20DI4653 v1.0.2.0  [SS1 -> X20TB32g.SS; SL -> X20BM12g.SL1]
  Supervision = off
X20DI4653h : X20DI4653 v1.0.2.0  [SS1 -> X20TB32h.SS; SL -> X20BM12h.SL1]
  Supervision = off
X20DI4653i : X20DI4653 v1.0.2.0  [SS1 -> X20TB32i.SS; SL -> X20BM12i.SL1]
  Supervision = off
X20DI4653j : X20DI4653 v1.0.2.0  [SS1 -> X20TB32j.SS; SL -> X20BM12j.SL1]
  Supervision = off
X20DO6639 : X20DO6639 v1.0.1.0  [SS1 -> X20TB32k.SS; SL -> X20BM12k.SL1]
  Supervision = off
X20DO6639a : X20DO6639 v1.0.1.0  [SS1 -> X20TB32l.SS; SL -> X20BM12l.SL1]
  Supervision = off
X20DO6639b : X20DO6639 v1.0.1.0  [SS1 -> X20TB32m.SS; SL -> X20BM12m.SL1]
  Supervision = off
X20DO6639c : X20DO6639 v1.0.1.0  [SS1 -> X20TB32n.SS; SL -> X20BM12n.SL1]
  Supervision = off
X20DO6639d : X20DO6639 v1.0.1.0  [SS1 -> X20TB32o.SS; SL -> X20BM12o.SL1]
  Supervision = off
X20DO6639e : X20DO6639 v1.0.1.0  [SS1 -> X20TB32p.SS; SL -> X20BM12p.SL1]
  Supervision = off
X20DO6639f : X20DO6639 v1.0.1.0  [SS1 -> X20TB32q.SS; SL -> X20BM12q.SL1]
  Supervision = off
X20DO6639g : X20DO6639 v1.0.1.0  [SS1 -> X20TB32r.SS; SL -> X20BM12r.SL1]
  Supervision = off
X20DO6639h : X20DO6639 v1.0.1.0  [SS1 -> X20TB32s.SS; SL -> X20BM12s.SL1]
  Supervision = off
X20DO6639i : X20DO6639 v1.0.1.0  [SS1 -> X20TB32t.SS; SL -> X20BM12t.SL1]
  Supervision = off
X20DO6639j : X20DO6639 v1.0.1.0  [SS1 -> X20TB32u.SS; SL -> X20BM12u.SL1]
  Supervision = off
X20DO6639k : X20DO6639 v1.0.1.0  [SS1 -> X20TB32v.SS; SL -> X20BM12v.SL1]
  Supervision = off
X20PS3300 : X20PS3300 v1.1.0.0  [SS1 -> X20TB12e.SS; SL -> X20BM01.SL1]
  Supervision = off
X20PS3300a : X20PS3300 v1.1.0.0  [SS1 -> X20TB12f.SS; SL -> X20BM01a.SL1]
  Supervision = off
X20TB12 : X20TB12 v1.0.0.0
X20TB12a : X20TB12 v1.0.0.0
X20TB12b : X20TB12 v1.0.0.0
X20TB12c : X20TB12 v1.0.0.0
X20TB12d : X20TB12 v1.0.0.0
X20TB12e : X20TB12 v1.0.0.0
X20TB12f : X20TB12 v1.0.0.0
X20TB32 : X20TB32 v1.0.0.1
X20TB32a : X20TB32 v1.0.0.1
X20TB32b : X20TB32 v1.0.0.1
X20TB32c : X20TB32 v1.0.0.1
X20TB32d : X20TB32 v1.0.0.1
X20TB32e : X20TB32 v1.0.0.1
X20TB32f : X20TB32 v1.0.0.1
X20TB32g : X20TB32 v1.0.0.1
X20TB32h : X20TB32 v1.0.0.1
X20TB32i : X20TB32 v1.0.0.1
X20TB32j : X20TB32 v1.0.0.1
X20TB32k : X20TB32 v1.0.0.1
X20TB32l : X20TB32 v1.0.0.1
X20TB32m : X20TB32 v1.0.0.1
X20TB32n : X20TB32 v1.0.0.1
X20TB32o : X20TB32 v1.0.0.1
X20TB32p : X20TB32 v1.0.0.1
X20TB32q : X20TB32 v1.0.0.1
X20TB32r : X20TB32 v1.0.0.1
X20TB32s : X20TB32 v1.0.0.1
X20TB32t : X20TB32 v1.0.0.1
X20TB32u : X20TB32 v1.0.0.1
X20TB32v : X20TB32 v1.0.0.1
```

### IoMap.iom - X20CP1584/IoMap.iom
```iecst
VAR_CONFIG
	Cyclic#2.::ProcessorJogFwd AT %IX."X20DI4653a".DigitalInput01;
	Cyclic#2.::ProcessorJogRev AT %IX."X20DI4653a".DigitalInput02;
	Cyclic#1.::EStopClear AT %IX."X20DI4653a".DigitalInput04;
	Cyclic#1.::ElectricDriveEnable AT %QX."X20CM8281".DigitalOutput01;
	Cyclic#1.::ActualDAC1 AT %QW."X20CM8281".AnalogOutput01;
	Cyclic#1.::ProcessorEncoderReset AT %QX."X20DC137A".Encoder01Reset;
	Cyclic#2.::CoilLineRun AT %IX."X20DI4653".DigitalInput01;
	Cyclic#1.ProcessorDriveReady AT %IX."X20CM8281".DigitalInput01;
	Cyclic#2.CoilLineReset AT %IX."X20DI4653".DigitalInput03;
	Cyclic#2.::MatlAtMeasureRoll AT %IX."X20DI4653a".DigitalInput03;
	Cyclic#2.::CoilLineHalt AT %IX."X20DI4653".DigitalInput02;
	::PowerOn AT %IX."X20DI4653".DigitalInput04;
	Cyclic#2.::CoilLineRunIndicator AT %QX."X20DO6639".DigitalOutput01;
	Cyclic#2.::CoilLineHaltIndicator AT %QX."X20DO6639".DigitalOutput02;
	Cyclic#2.::ShearValve AT %QX."X20DO6639".DigitalOutput04;
	::LTValve AT %QX."X20DO6639a".DigitalOutput01;
	::VValve AT %QX."X20DO6639a".DigitalOutput02;
	::LHoleValve AT %QX."X20DO6639a".DigitalOutput03;
	LevelerBrakeSolenoid AT %QX."X20DO6639a".DigitalOutput06;
	Cyclic#2.PunchMasterShiftSolenoid AT %QX."X20DO6639b".DigitalOutput01;
	Cyclic#2.OutSideGuideSolenoid AT %QX."X20DO6639b".DigitalOutput02;
	Cyclic#2.FourFootCenterSolenoid AT %QX."X20DO6639b".DigitalOutput03;
	Cyclic#2.FiveFootCenterSolenoid AT %QX."X20DO6639b".DigitalOutput04;
	Cyclic#2.SixFootCenterSolenoid AT %QX."X20DO6639b".DigitalOutput05;
	Cyclic#2.FourFootOutsideSolenoid AT %QX."X20DO6639b".DigitalOutput06;
	Cyclic#2.FiveFootOutsideSolenoid AT %QX."X20DO6639c".DigitalOutput01;
	Cyclic#2.SixFootOutsideSolenoid AT %QX."X20DO6639c".DigitalOutput02;
	Cyclic#2.DamperHoleSolenoid AT %QX."X20DO6639c".DigitalOutput03;
	Cyclic#2.HolePunchSelectedSolenoid AT %QX."X20DO6639c".DigitalOutput04;
	Cyclic#2.DieSelectSolenoid AT %QX."X20DO6639c".DigitalOutput05;
	Cyclic#1.::ActlMetalEncoder AT %ID."X20DC137A".Encoder01;
	::BackGaugeJogInPB AT %IX."X20DI4653f".DigitalInput01;
	::BackGaugeJogOutPB AT %IX."X20DI4653f".DigitalInput02;
	::BackGaugeHomeLS AT %IX."X20DI4653f".DigitalInput03;
	FWBResetPB AT %IX."X20DI4653f".DigitalInput04;
	Cyclic#2.::HolePunchUp AT %IX."X20DI4653b".DigitalInput04;
	Cyclic#2.::LatchCylinderInSolenoid AT %QX."X20DO6639i".DigitalOutput01;
	Cyclic#2.::LatchCylinderOutSolenoid AT %QX."X20DO6639i".DigitalOutput02;
	Cyclic#2.::BrakeBeamRaise AT %QX."X20DO6639i".DigitalOutput03;
	Cyclic#2.::BrakeBeamLower AT %QX."X20DO6639i".DigitalOutput04;
	Cyclic#2.::FormHeadUpSolenoid AT %QX."X20DO6639i".DigitalOutput05;
	Cyclic#2.::BrakeStopsInSolenoid AT %QX."X20DO6639j".DigitalOutput01;
	Cyclic#2.::BrakeStopsOutSolenoid AT %QX."X20DO6639j".DigitalOutput02;
	Cyclic#2.::FormHeadDownSolenoid AT %QX."X20DO6639j".DigitalOutput04;
END_VAR
```

## Configuration E1000V2_1

### Task classes (Cpu.sw)
```
Cyclic#1 (cycle 1000 us, tolerance 0 us):
  EFdrHydDrv <- EFdrHydDrv.prg
  CEF <- CEF.prg
  IMotion2 <- IMotion2.prg
Cyclic#2 (cycle 20000 us, tolerance 20000 us):
  SysCheck <- SysCheck.prg
  E2Feeder <- E2Feeder.prg
  PMaster <- PMaster.prg
  Pinspotter <- Pinspotter.prg
  E_FWB <- E_FWB.prg
  DH800 <- DH800.prg
Cyclic#4 (cycle 100000 us, tolerance 100000 us):
  Server <- LibAsTCP1_ST.Server.prg
Binaries: TCData, arconfig, asfw, ashwd, iomap, User, Role, sysconf
Libraries: asstring, runtime, asieccon, standard, astime, astcp
```

### Hardware
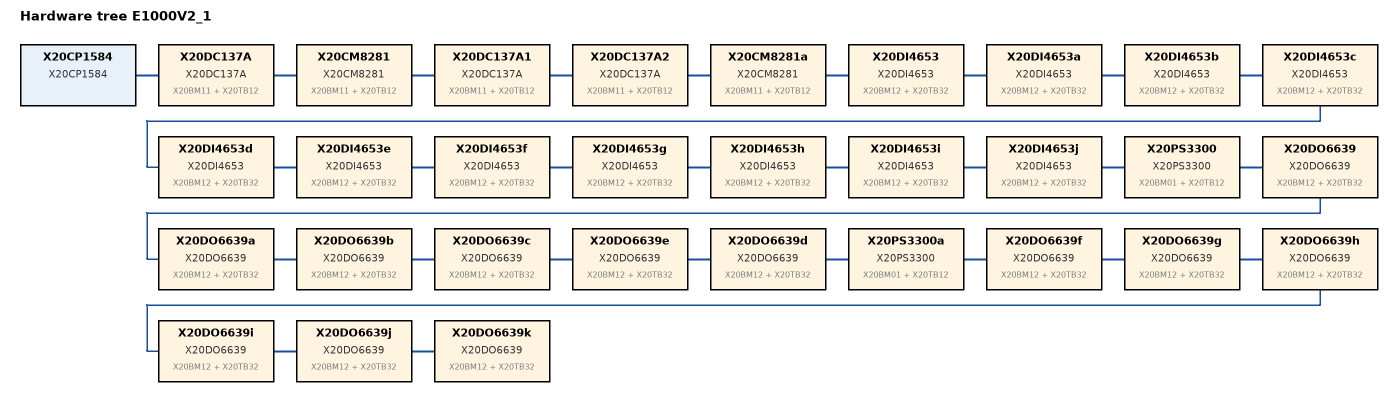
```
X20BM01 : X20BM01 v1.0.1.1  [X2X1 -> X20BM12j.X2X2]
X20BM01a : X20BM01 v1.0.1.1  [X2X1 -> X20BM12o.X2X2]
X20BM11 : X20BM11 v1.0.0.1  [X2X1 -> X20CP1584.IF6]
X20BM11a : X20BM11 v1.0.0.1  [X2X1 -> X20BM11.X2X2]
X20BM11b : X20BM11 v1.0.0.1  [X2X1 -> X20BM11a.X2X2]
X20BM11c : X20BM11 v1.0.0.1  [X2X1 -> X20BM11b.X2X2]
X20BM11d : X20BM11 v1.0.0.1  [X2X1 -> X20BM11c.X2X2]
X20BM12 : X20BM12 v1.0.0.1  [X2X1 -> X20BM11d.X2X2]
X20BM12a : X20BM12 v1.0.0.1  [X2X1 -> X20BM12.X2X2]
X20BM12b : X20BM12 v1.0.0.1  [X2X1 -> X20BM12a.X2X2]
X20BM12c : X20BM12 v1.0.0.1  [X2X1 -> X20BM12b.X2X2]
X20BM12d : X20BM12 v1.0.0.1  [X2X1 -> X20BM12c.X2X2]
X20BM12e : X20BM12 v1.0.0.1  [X2X1 -> X20BM12d.X2X2]
X20BM12f : X20BM12 v1.0.0.1  [X2X1 -> X20BM12e.X2X2]
X20BM12g : X20BM12 v1.0.0.1  [X2X1 -> X20BM12f.X2X2]
X20BM12h : X20BM12 v1.0.0.1  [X2X1 -> X20BM12g.X2X2]
X20BM12i : X20BM12 v1.0.0.1  [X2X1 -> X20BM12h.X2X2]
X20BM12j : X20BM12 v1.0.0.1  [X2X1 -> X20BM12i.X2X2]
X20BM12k : X20BM12 v1.0.0.1  [X2X1 -> X20BM01.X2X2]
X20BM12l : X20BM12 v1.0.0.1  [X2X1 -> X20BM12k.X2X2]
X20BM12m : X20BM12 v1.0.0.1  [X2X1 -> X20BM12l.X2X2]
X20BM12n : X20BM12 v1.0.0.1  [X2X1 -> X20BM12m.X2X2]
X20BM12o : X20BM12 v1.0.0.1  [X2X1 -> X20BM12p.X2X2]
X20BM12p : X20BM12 v1.0.0.1  [X2X1 -> X20BM12n.X2X2]
X20BM12q : X20BM12 v1.0.0.1  [X2X1 -> X20BM01a.X2X2]
X20BM12r : X20BM12 v1.0.0.1  [X2X1 -> X20BM12q.X2X2]
X20BM12s : X20BM12 v1.0.0.1  [X2X1 -> X20BM12r.X2X2]
X20BM12t : X20BM12 v1.0.0.1  [X2X1 -> X20BM12s.X2X2]
X20BM12u : X20BM12 v1.0.0.1  [X2X1 -> X20BM12t.X2X2]
X20BM12v : X20BM12 v1.0.0.1  [X2X1 -> X20BM12u.X2X2]
X20CM8281 : X20CM8281 v1.0.4.0  [SS1 -> X20TB12a.SS; SL -> X20BM11a.SL1]
  Supervision = off
X20CM8281a : X20CM8281 v1.0.4.0  [SS1 -> X20TB12d.SS; SL -> X20BM11d.SL1]
  Supervision = off
X20CP1584 : X20CP1584 v1.3.0.0
  Connector IF2:
    ActivateDevice = 1
    EthInterfaceRedundant = 0
    Mode = Manual
    InternetAddress = 10.1.254.101
  Connector IF3:
    EplInterfaceRedundant = 0
    EplEthInterfaceRedundant = 0
  Connector IF6:
    CycleTime = 1000
  ConfigurationID = X20_CPU_E1000
  EnableUsbRemoteInstall = 1
  TimerDeviceType = EPLX2X
  TimerDevice = X20CP1584.IF6
  Cyclic1Duration = 1000
  Cyclic1Tolerance = 0
  Cyclic1Output = 1
  Cyclic2Duration = 20000
  Cyclic2Tolerance = 20000
  Cyclic3Duration = 50000
  Cyclic3Tolerance = 50000
  Cyclic4Duration = 100000
  Cyclic4Tolerance = 100000
  Cyclic5Duration = 200000
  Cyclic5Tolerance = 200000
  Cyclic6Duration = 500000
  Cyclic6Tolerance = 500000
  Cyclic7Duration = 1000000
  Cyclic7Tolerance = 1000000
  Cyclic8Duration = 10000
  Cyclic8Tolerance = 30000000
  Route1
X20DC137A : X20DC137A v1.0.0.3  [SS1 -> X20TB12.SS; SL -> X20BM11.SL1]
  Supervision = off
  CounterStd01 = 32Bit
  BWConfigChannel03 = off
X20DC137A1 : X20DC137A v1.0.0.3  [SS1 -> X20TB12b.SS; SL -> X20BM11b.SL1]
  Supervision = off
  CounterStd01 = 32Bit
  BWConfigChannel03 = off
X20DC137A2 : X20DC137A v1.0.0.3  [SS1 -> X20TB12c.SS; SL -> X20BM11c.SL1]
  Supervision = off
  CounterStd01 = 32Bit
  BWConfigChannel03 = off
X20DI4653 : X20DI4653 v1.0.2.0  [SS1 -> X20TB32.SS; SL -> X20BM12.SL1]
  Supervision = off
X20DI4653a : X20DI4653 v1.0.2.0  [SS1 -> X20TB32a.SS; SL -> X20BM12a.SL1]
  Supervision = off
X20DI4653b : X20DI4653 v1.0.2.0  [SS1 -> X20TB32b.SS; SL -> X20BM12b.SL1]
  Supervision = off
X20DI4653c : X20DI4653 v1.0.2.0  [SS1 -> X20TB32c.SS; SL -> X20BM12c.SL1]
  Supervision = off
X20DI4653d : X20DI4653 v1.0.2.0  [SS1 -> X20TB32d.SS; SL -> X20BM12d.SL1]
  Supervision = off
X20DI4653e : X20DI4653 v1.0.2.0  [SS1 -> X20TB32e.SS; SL -> X20BM12e.SL1]
  Supervision = off
X20DI4653f : X20DI4653 v1.0.2.0  [SS1 -> X20TB32f.SS; SL -> X20BM12f.SL1]
  Supervision = off
X20DI4653g : X20DI4653 v1.0.2.0  [SS1 -> X20TB32g.SS; SL -> X20BM12g.SL1]
  Supervision = off
X20DI4653h : X20DI4653 v1.0.2.0  [SS1 -> X20TB32h.SS; SL -> X20BM12h.SL1]
  Supervision = off
X20DI4653i : X20DI4653 v1.0.2.0  [SS1 -> X20TB32i.SS; SL -> X20BM12i.SL1]
  Supervision = off
X20DI4653j : X20DI4653 v1.0.2.0  [SS1 -> X20TB32j.SS; SL -> X20BM12j.SL1]
  Supervision = off
X20DO6639 : X20DO6639 v1.0.1.0  [SS1 -> X20TB32k.SS; SL -> X20BM12k.SL1]
  Supervision = off
X20DO6639a : X20DO6639 v1.0.1.0  [SS1 -> X20TB32l.SS; SL -> X20BM12l.SL1]
  Supervision = off
X20DO6639b : X20DO6639 v1.0.1.0  [SS1 -> X20TB32m.SS; SL -> X20BM12m.SL1]
  Supervision = off
X20DO6639c : X20DO6639 v1.0.1.0  [SS1 -> X20TB32n.SS; SL -> X20BM12n.SL1]
  Supervision = off
X20DO6639d : X20DO6639 v1.0.1.0  [SS1 -> X20TB32o.SS; SL -> X20BM12o.SL1]
  Supervision = off
X20DO6639e : X20DO6639 v1.0.1.0  [SS1 -> X20TB32p.SS; SL -> X20BM12p.SL1]
  Supervision = off
X20DO6639f : X20DO6639 v1.0.1.0  [SS1 -> X20TB32q.SS; SL -> X20BM12q.SL1]
  Supervision = off
X20DO6639g : X20DO6639 v1.0.1.0  [SS1 -> X20TB32r.SS; SL -> X20BM12r.SL1]
  Supervision = off
X20DO6639h : X20DO6639 v1.0.1.0  [SS1 -> X20TB32s.SS; SL -> X20BM12s.SL1]
  Supervision = off
X20DO6639i : X20DO6639 v1.0.1.0  [SS1 -> X20TB32t.SS; SL -> X20BM12t.SL1]
  Supervision = off
X20DO6639j : X20DO6639 v1.0.1.0  [SS1 -> X20TB32u.SS; SL -> X20BM12u.SL1]
  Supervision = off
X20DO6639k : X20DO6639 v1.0.1.0  [SS1 -> X20TB32v.SS; SL -> X20BM12v.SL1]
  Supervision = off
X20PS3300 : X20PS3300 v1.1.0.0  [SS1 -> X20TB12e.SS; SL -> X20BM01.SL1]
  Supervision = off
X20PS3300a : X20PS3300 v1.1.0.0  [SS1 -> X20TB12f.SS; SL -> X20BM01a.SL1]
  Supervision = off
X20TB12 : X20TB12 v1.0.0.0
X20TB12a : X20TB12 v1.0.0.0
X20TB12b : X20TB12 v1.0.0.0
X20TB12c : X20TB12 v1.0.0.0
X20TB12d : X20TB12 v1.0.0.0
X20TB12e : X20TB12 v1.0.0.0
X20TB12f : X20TB12 v1.0.0.0
X20TB32 : X20TB32 v1.0.0.1
X20TB32a : X20TB32 v1.0.0.1
X20TB32b : X20TB32 v1.0.0.1
X20TB32c : X20TB32 v1.0.0.1
X20TB32d : X20TB32 v1.0.0.1
X20TB32e : X20TB32 v1.0.0.1
X20TB32f : X20TB32 v1.0.0.1
X20TB32g : X20TB32 v1.0.0.1
X20TB32h : X20TB32 v1.0.0.1
X20TB32i : X20TB32 v1.0.0.1
X20TB32j : X20TB32 v1.0.0.1
X20TB32k : X20TB32 v1.0.0.1
X20TB32l : X20TB32 v1.0.0.1
X20TB32m : X20TB32 v1.0.0.1
X20TB32n : X20TB32 v1.0.0.1
X20TB32o : X20TB32 v1.0.0.1
X20TB32p : X20TB32 v1.0.0.1
X20TB32q : X20TB32 v1.0.0.1
X20TB32r : X20TB32 v1.0.0.1
X20TB32s : X20TB32 v1.0.0.1
X20TB32t : X20TB32 v1.0.0.1
X20TB32u : X20TB32 v1.0.0.1
X20TB32v : X20TB32 v1.0.0.1
```
